IF initializeEvents THEN 
	initializeEvents := FALSE; 
	Emergency_zone_1.CreateEx(TC_Events.Kremer_Events.Emergency_zone_1, TRUE, 0); 
	Emergency_zone_2.CreateEx(TC_Events.Kremer_Events.Emergency_zone_2, TRUE, 0); 
	Emergency_zone_3.CreateEx(TC_Events.Kremer_Events.Emergency_zone_3, TRUE, 0); 
	Emergency_zone_4.CreateEx(TC_Events.Kremer_Events.Emergency_zone_4, TRUE, 0); 
	Emergency_zone_5.CreateEx(TC_Events.Kremer_Events.Emergency_zone_5, TRUE, 0); 
	Emergency_zone_6.CreateEx(TC_Events.Kremer_Events.Emergency_zone_6, TRUE, 0); 
	Emergency_zone_7.CreateEx(TC_Events.Kremer_Events.Emergency_zone_7, TRUE, 0); 
	In_mold_drying_emergency_stop_pressed_front_side.CreateEx(TC_Events.Kremer_Events.In_mold_drying_emergency_stop_pressed_front_side, TRUE, 0); 
	In_mold_drying_emergency_stop_pressed_back_side.CreateEx(TC_Events.Kremer_Events.In_mold_drying_emergency_stop_pressed_back_side, TRUE, 0); 
	In_mold_drying_door_opend_frontside_left.CreateEx(TC_Events.Kremer_Events.In_mold_drying_door_opend_frontside_left, TRUE, 0); 
	In_mold_drying_door_opened_frontside_middle.CreateEx(TC_Events.Kremer_Events.In_mold_drying_door_opened_frontside_middle, TRUE, 0); 
	In_mold_drying_door_opened_frontside_right.CreateEx(TC_Events.Kremer_Events.In_mold_drying_door_opened_frontside_right, TRUE, 0); 
	In_mold_drying_double_door_opened_backside_left_1.CreateEx(TC_Events.Kremer_Events.In_mold_drying_double_door_opened_backside_left_1, TRUE, 0); 
	In_mold_drying_double_door_opened_backside_left_2.CreateEx(TC_Events.Kremer_Events.In_mold_drying_double_door_opened_backside_left_2, TRUE, 0); 
	In_mold_drying_double_door_opened_backside_Middle_1.CreateEx(TC_Events.Kremer_Events.In_mold_drying_double_door_opened_backside_Middle_1, TRUE, 0); 
	In_mold_drying_double_door_opened_backside_Middle_2.CreateEx(TC_Events.Kremer_Events.In_mold_drying_double_door_opened_backside_Middle_2, TRUE, 0); 
	In_mold_drying_double_door_opened_backside_Right_1.CreateEx(TC_Events.Kremer_Events.In_mold_drying_double_door_opened_backside_Right_1, TRUE, 0); 
	In_mold_drying_double_door_opened_backside_Right_2.CreateEx(TC_Events.Kremer_Events.In_mold_drying_double_door_opened_backside_Right_2, TRUE, 0); 
	Gantry_A_front_door_openend_right.CreateEx(TC_Events.Kremer_Events.Gantry_A_front_door_openend_right, TRUE, 0); 
	Gantry_A_front_door_openend_left.CreateEx(TC_Events.Kremer_Events.Gantry_A_front_door_openend_left, TRUE, 0); 
	Gantry_A_Back_door_openend.CreateEx(TC_Events.Kremer_Events.Gantry_A_Back_door_openend, TRUE, 0); 
	Gantry_B_front_door_openend_left.CreateEx(TC_Events.Kremer_Events.Gantry_B_front_door_openend_left, TRUE, 0); 
	Gantry_B_front_door_openend_right.CreateEx(TC_Events.Kremer_Events.Gantry_B_front_door_openend_right, TRUE, 0); 
	Gantry_B_Back_door_openend.CreateEx(TC_Events.Kremer_Events.Gantry_B_Back_door_openend, TRUE, 0); 
	Emergency_stop_pressed_Gantry_A_backside.CreateEx(TC_Events.Kremer_Events.Emergency_stop_pressed_Gantry_A_backside, TRUE, 0); 
	Emergency_stop_pressed_Gantry_A_Frontside.CreateEx(TC_Events.Kremer_Events.Emergency_stop_pressed_Gantry_A_Frontside, TRUE, 0); 
	Emergency_stop_pressed_Gantry_B_Backside.CreateEx(TC_Events.Kremer_Events.Emergency_stop_pressed_Gantry_B_Backside, TRUE, 0); 
	Emergency_stop_pressed_Gantry_B_Frontside.CreateEx(TC_Events.Kremer_Events.Emergency_stop_pressed_Gantry_B_Frontside, TRUE, 0); 
	_24_volt_circuit_in_error_1.CreateEx(TC_Events.Kremer_Events._24_volt_circuit_in_error_1, TRUE, 0); 
	_24_volt_circuit_in_error_2.CreateEx(TC_Events.Kremer_Events._24_volt_circuit_in_error_2, TRUE, 0); 
	No_product_loaded_please_load_a_valid_product_first.CreateEx(TC_Events.Kremer_Events.No_product_loaded_please_load_a_valid_product_first, TRUE, 0); 
	Main_air_supply_has_an_error.CreateEx(TC_Events.Kremer_Events.Main_air_supply_has_an_error, TRUE, 0); 
	In_mold_drying_hydraulic_pump_softstarter_failure.CreateEx(TC_Events.Kremer_Events.In_mold_drying_hydraulic_pump_softstarter_failure, TRUE, 0); 
	In_mold_drying_hydraulic_pump_maintenance_switch.CreateEx(TC_Events.Kremer_Events.In_mold_drying_hydraulic_pump_maintenance_switch, TRUE, 0); 
	In_mold_drying_cooling_fan_thermal_failure.CreateEx(TC_Events.Kremer_Events.In_mold_drying_cooling_fan_thermal_failure, TRUE, 0); 
	In_mold_drying_cooling_fan_maintenance_switch.CreateEx(TC_Events.Kremer_Events.In_mold_drying_cooling_fan_maintenance_switch, TRUE, 0); 
	In_mold_drying_filter_motor_thermal.CreateEx(TC_Events.Kremer_Events.In_mold_drying_filter_motor_thermal, TRUE, 0); 
	In_mold_drying_filter_motor_maintenance.CreateEx(TC_Events.Kremer_Events.In_mold_drying_filter_motor_maintenance, TRUE, 0); 
	Css_has_an_active_error.CreateEx(TC_Events.Kremer_Events.Css_has_an_active_error, TRUE, 0); 
	Both_Pulp_Tanks_below_Low_Level_stopping_IMD.CreateEx(TC_Events.Kremer_Events.Both_Pulp_Tanks_below_Low_Level_stopping_IMD, TRUE, 0); 
	RHSR_Bottom_mold_A_moving_while_top_mold_A_not_in_position.CreateEx(TC_Events.Kremer_Events.RHSR_Bottom_mold_A_moving_while_top_mold_A_not_in_position, TRUE, 0); 
	RHSR_Bottom_mold_A_moving_while_transfer_mold_A_not_in_position.CreateEx(TC_Events.Kremer_Events.RHSR_Bottom_mold_A_moving_while_transfer_mold_A_not_in_position, TRUE, 0); 
	RHSR_Bottom_mold_B_moving_while_top_mold_B_not_in_position.CreateEx(TC_Events.Kremer_Events.RHSR_Bottom_mold_B_moving_while_top_mold_B_not_in_position, TRUE, 0); 
	RHSR_Bottom_mold_B_moving_while_transfer_mold_B_not_in_position.CreateEx(TC_Events.Kremer_Events.RHSR_Bottom_mold_B_moving_while_transfer_mold_B_not_in_position, TRUE, 0); 
	RHSR_Takeout_A_moving_while_vertical_cylinder_is_not_down.CreateEx(TC_Events.Kremer_Events.RHSR_Takeout_A_moving_while_vertical_cylinder_is_not_down, TRUE, 0); 
	RHSR_Takeout_B_moving_while_vertical_cylinder_is_not_down.CreateEx(TC_Events.Kremer_Events.RHSR_Takeout_B_moving_while_vertical_cylinder_is_not_down, TRUE, 0); 
	RHSR_TopMold_A_moving_while_bottom_mold_A_is_not_in_position.CreateEx(TC_Events.Kremer_Events.RHSR_TopMold_A_moving_while_bottom_mold_A_is_not_in_position, TRUE, 0); 
	RHSR_TopMold_B_moving_while_bottom_mold_B_is_not_in_position.CreateEx(TC_Events.Kremer_Events.RHSR_TopMold_B_moving_while_bottom_mold_B_is_not_in_position, TRUE, 0); 
	RHSR_Transfermold_moving_while_bottom_mold_A_is_not_in_posititon.CreateEx(TC_Events.Kremer_Events.RHSR_Transfermold_moving_while_bottom_mold_A_is_not_in_posititon, TRUE, 0); 
	RHSR_Transfermold_moving_while_bottom_mold_B_is_not_in_position.CreateEx(TC_Events.Kremer_Events.RHSR_Transfermold_moving_while_bottom_mold_B_is_not_in_position, TRUE, 0); 
	RHSR_Transfermold_moving_while_spraybar_is_not_at_one_of_rest_positions.CreateEx(TC_Events.Kremer_Events.RHSR_Transfermold_moving_while_spraybar_is_not_at_one_of_rest_positions, TRUE, 0); 
	Temperature_difference_between_top_and_bottom_mold_side_A_to_high.CreateEx(TC_Events.Kremer_Events.Temperature_difference_between_top_and_bottom_mold_side_A_to_high, TRUE, 0); 
	Temperature_difference_between_top_and_bottom_mold_side_B_to_high.CreateEx(TC_Events.Kremer_Events.Temperature_difference_between_top_and_bottom_mold_side_B_to_high, TRUE, 0); 
	Spare56.CreateEx(TC_Events.Kremer_Events.Spare56, TRUE, 0); 
	Auxiliary_filter_100_dirty.CreateEx(TC_Events.Kremer_Events.Auxiliary_filter_100_dirty, TRUE, 0); 
	Auxiliary_filter_75_dirty.CreateEx(TC_Events.Kremer_Events.Auxiliary_filter_75_dirty, TRUE, 0); 
	Oil_filter_100_dirty.CreateEx(TC_Events.Kremer_Events.Oil_filter_100_dirty, TRUE, 0); 
	Oil_filter_75_dirty.CreateEx(TC_Events.Kremer_Events.Oil_filter_75_dirty, TRUE, 0); 
	Fan_on_MCC2_error.CreateEx(TC_Events.Kremer_Events.Fan_on_MCC2_error, TRUE, 0); 
	_24V_error_on_MCC2.CreateEx(TC_Events.Kremer_Events._24V_error_on_MCC2, TRUE, 0); 
	Oil_temperature_too_low.CreateEx(TC_Events.Kremer_Events.Oil_temperature_too_low, TRUE, 0); 
	Oil_temperature_too_high.CreateEx(TC_Events.Kremer_Events.Oil_temperature_too_high, TRUE, 0); 
	Top_mold_A_error_on_balluf.CreateEx(TC_Events.Kremer_Events.Top_mold_A_error_on_balluf, TRUE, 0); 
	Top_mold_A_position_error.CreateEx(TC_Events.Kremer_Events.Top_mold_A_position_error, TRUE, 0); 
	Top_mold_A_timed_out_Did_not_reach_bottommold_position_in_time.CreateEx(TC_Events.Kremer_Events.Top_mold_A_timed_out_Did_not_reach_bottommold_position_in_time, TRUE, 0); 
	Top_mold_A_Rod_side_pressure_too_high.CreateEx(TC_Events.Kremer_Events.Top_mold_A_Rod_side_pressure_too_high, TRUE, 0); 
	Top_mold_A_Bot_side_pressure_too_high.CreateEx(TC_Events.Kremer_Events.Top_mold_A_Bot_side_pressure_too_high, TRUE, 0); 
	Topmold_A_heating_zone_1_connector_not_connected.CreateEx(TC_Events.Kremer_Events.Topmold_A_heating_zone_1_connector_not_connected, TRUE, 0); 
	Topmold_A_heating_zone_1_PT100_wrong_position.CreateEx(TC_Events.Kremer_Events.Topmold_A_heating_zone_1_PT100_wrong_position, TRUE, 0); 
	Topmold_A_heating_zone_1_PT100_loose.CreateEx(TC_Events.Kremer_Events.Topmold_A_heating_zone_1_PT100_loose, TRUE, 0); 
	Topmold_A_heating_zone_1_PT100_not_inserted.CreateEx(TC_Events.Kremer_Events.Topmold_A_heating_zone_1_PT100_not_inserted, TRUE, 0); 
	Topmold_A_heating_zone_1_Temperature_above_setpoint.CreateEx(TC_Events.Kremer_Events.Topmold_A_heating_zone_1_Temperature_above_setpoint, TRUE, 0); 
	Topmold_A_heating_zone_1_Temperature_below_setpoint.CreateEx(TC_Events.Kremer_Events.Topmold_A_heating_zone_1_Temperature_below_setpoint, TRUE, 0); 
	Topmold_A_heating_zone_1_PT100_wirebreak.CreateEx(TC_Events.Kremer_Events.Topmold_A_heating_zone_1_PT100_wirebreak, TRUE, 0); 
	Topmold_A_heating_zone_1_Thermal.CreateEx(TC_Events.Kremer_Events.Topmold_A_heating_zone_1_Thermal, TRUE, 0); 
	Topmold_A_heating_zone_1_temperature_above_250_degree_heating_element_switched_off.CreateEx(TC_Events.Kremer_Events.Topmold_A_heating_zone_1_temperature_above_250_degree_heating_element_switched_off, TRUE, 0); 
	Topmold_A_heating_zone_1_temperature_above_230_degree.CreateEx(TC_Events.Kremer_Events.Topmold_A_heating_zone_1_temperature_above_230_degree, TRUE, 0); 
	Topmold_A_heating_zone_2_connector_not_connected.CreateEx(TC_Events.Kremer_Events.Topmold_A_heating_zone_2_connector_not_connected, TRUE, 0); 
	Topmold_A_heating_zone_2_PT100_wrong_position.CreateEx(TC_Events.Kremer_Events.Topmold_A_heating_zone_2_PT100_wrong_position, TRUE, 0); 
	Topmold_A_heating_zone_2_PT100_loose.CreateEx(TC_Events.Kremer_Events.Topmold_A_heating_zone_2_PT100_loose, TRUE, 0); 
	Topmold_A_heating_zone_2_PT100_not_inserted.CreateEx(TC_Events.Kremer_Events.Topmold_A_heating_zone_2_PT100_not_inserted, TRUE, 0); 
	Topmold_A_heating_zone_2_Temperature_above_setpoint.CreateEx(TC_Events.Kremer_Events.Topmold_A_heating_zone_2_Temperature_above_setpoint, TRUE, 0); 
	Topmold_A_heating_zone_2_Temperature_below_setpoint.CreateEx(TC_Events.Kremer_Events.Topmold_A_heating_zone_2_Temperature_below_setpoint, TRUE, 0); 
	Topmold_A_heating_zone_2_PT100_wirebreak.CreateEx(TC_Events.Kremer_Events.Topmold_A_heating_zone_2_PT100_wirebreak, TRUE, 0); 
	Topmold_A_heating_zone_2_Thermal.CreateEx(TC_Events.Kremer_Events.Topmold_A_heating_zone_2_Thermal, TRUE, 0); 
	Topmold_A_heating_zone_2_temperature_above_250_degree_heating_element_switched_off.CreateEx(TC_Events.Kremer_Events.Topmold_A_heating_zone_2_temperature_above_250_degree_heating_element_switched_off, TRUE, 0); 
	Topmold_A_heating_zone_2_temperature_above_230_degree.CreateEx(TC_Events.Kremer_Events.Topmold_A_heating_zone_2_temperature_above_230_degree, TRUE, 0); 
	Tranfermold_timed_out_did_not_reach_bottommold_position_in_time.CreateEx(TC_Events.Kremer_Events.Tranfermold_timed_out_did_not_reach_bottommold_position_in_time, TRUE, 0); 
	Tranfermold_timed_out_did_not_reach_forming_position_in_time.CreateEx(TC_Events.Kremer_Events.Tranfermold_timed_out_did_not_reach_forming_position_in_time, TRUE, 0); 
	Topmold_A_heating_zone_3_connector_not_connected.CreateEx(TC_Events.Kremer_Events.Topmold_A_heating_zone_3_connector_not_connected, TRUE, 0); 
	Topmold_A_heating_zone_3_PT100_wrong_position.CreateEx(TC_Events.Kremer_Events.Topmold_A_heating_zone_3_PT100_wrong_position, TRUE, 0); 
	Topmold_A_heating_zone_3_PT100_loose.CreateEx(TC_Events.Kremer_Events.Topmold_A_heating_zone_3_PT100_loose, TRUE, 0); 
	Topmold_A_heating_zone_3_PT100_not_inserted.CreateEx(TC_Events.Kremer_Events.Topmold_A_heating_zone_3_PT100_not_inserted, TRUE, 0); 
	Topmold_A_heating_zone_3_Temperature_above_setpoint.CreateEx(TC_Events.Kremer_Events.Topmold_A_heating_zone_3_Temperature_above_setpoint, TRUE, 0); 
	Topmold_A_heating_zone_3_Temperature_below_setpoint.CreateEx(TC_Events.Kremer_Events.Topmold_A_heating_zone_3_Temperature_below_setpoint, TRUE, 0); 
	Topmold_A_heating_zone_3_PT100_wirebreak.CreateEx(TC_Events.Kremer_Events.Topmold_A_heating_zone_3_PT100_wirebreak, TRUE, 0); 
	Topmold_A_heating_zone_3_Thermal.CreateEx(TC_Events.Kremer_Events.Topmold_A_heating_zone_3_Thermal, TRUE, 0); 
	Topmold_A_heating_zone_3_temperature_above_250_degree_heating_element_switched_off.CreateEx(TC_Events.Kremer_Events.Topmold_A_heating_zone_3_temperature_above_250_degree_heating_element_switched_off, TRUE, 0); 
	Topmold_A_heating_zone_3_temperature_above_230_degree.CreateEx(TC_Events.Kremer_Events.Topmold_A_heating_zone_3_temperature_above_230_degree, TRUE, 0); 
	Topmold_A_heating_zone_4_connector_not_connected.CreateEx(TC_Events.Kremer_Events.Topmold_A_heating_zone_4_connector_not_connected, TRUE, 0); 
	Topmold_A_heating_zone_4_PT100_wrong_position.CreateEx(TC_Events.Kremer_Events.Topmold_A_heating_zone_4_PT100_wrong_position, TRUE, 0); 
	Topmold_A_heating_zone_4_PT100_loose.CreateEx(TC_Events.Kremer_Events.Topmold_A_heating_zone_4_PT100_loose, TRUE, 0); 
	Topmold_A_heating_zone_4_PT100_not_inserted.CreateEx(TC_Events.Kremer_Events.Topmold_A_heating_zone_4_PT100_not_inserted, TRUE, 0); 
	Topmold_A_heating_zone_4_Temperature_above_setpoint.CreateEx(TC_Events.Kremer_Events.Topmold_A_heating_zone_4_Temperature_above_setpoint, TRUE, 0); 
	Topmold_A_heating_zone_4_Temperature_below_setpoint.CreateEx(TC_Events.Kremer_Events.Topmold_A_heating_zone_4_Temperature_below_setpoint, TRUE, 0); 
	Topmold_A_heating_zone_4_PT100_wirebreak.CreateEx(TC_Events.Kremer_Events.Topmold_A_heating_zone_4_PT100_wirebreak, TRUE, 0); 
	Topmold_A_heating_zone_4_Thermal.CreateEx(TC_Events.Kremer_Events.Topmold_A_heating_zone_4_Thermal, TRUE, 0); 
	Topmold_A_heating_zone_4_temperature_above_250_degree_heating_element_switched_off.CreateEx(TC_Events.Kremer_Events.Topmold_A_heating_zone_4_temperature_above_250_degree_heating_element_switched_off, TRUE, 0); 
	Topmold_A_heating_zone_4_temperature_above_230_degree.CreateEx(TC_Events.Kremer_Events.Topmold_A_heating_zone_4_temperature_above_230_degree, TRUE, 0); 
	Topmold_A_heating_zone_5_connector_not_connected.CreateEx(TC_Events.Kremer_Events.Topmold_A_heating_zone_5_connector_not_connected, TRUE, 0); 
	Topmold_A_heating_zone_5_PT100_wrong_position.CreateEx(TC_Events.Kremer_Events.Topmold_A_heating_zone_5_PT100_wrong_position, TRUE, 0); 
	Topmold_A_heating_zone_5_PT100_loose.CreateEx(TC_Events.Kremer_Events.Topmold_A_heating_zone_5_PT100_loose, TRUE, 0); 
	Topmold_A_heating_zone_5_PT100_not_inserted.CreateEx(TC_Events.Kremer_Events.Topmold_A_heating_zone_5_PT100_not_inserted, TRUE, 0); 
	Topmold_A_heating_zone_5_Temperature_above_setpoint.CreateEx(TC_Events.Kremer_Events.Topmold_A_heating_zone_5_Temperature_above_setpoint, TRUE, 0); 
	Topmold_A_heating_zone_5_Temperature_below_setpoint.CreateEx(TC_Events.Kremer_Events.Topmold_A_heating_zone_5_Temperature_below_setpoint, TRUE, 0); 
	Topmold_A_heating_zone_5_PT100_wirebreak.CreateEx(TC_Events.Kremer_Events.Topmold_A_heating_zone_5_PT100_wirebreak, TRUE, 0); 
	Topmold_A_heating_zone_5_Thermal.CreateEx(TC_Events.Kremer_Events.Topmold_A_heating_zone_5_Thermal, TRUE, 0); 
	Topmold_A_heating_zone_5_temperature_above_250_degree_heating_element_switched_off.CreateEx(TC_Events.Kremer_Events.Topmold_A_heating_zone_5_temperature_above_250_degree_heating_element_switched_off, TRUE, 0); 
	Topmold_A_heating_zone_5_temperature_above_230_degree.CreateEx(TC_Events.Kremer_Events.Topmold_A_heating_zone_5_temperature_above_230_degree, TRUE, 0); 
	Topmold_A_heating_zone_6_connector_not_connected.CreateEx(TC_Events.Kremer_Events.Topmold_A_heating_zone_6_connector_not_connected, TRUE, 0); 
	Topmold_A_heating_zone_6_PT100_wrong_position.CreateEx(TC_Events.Kremer_Events.Topmold_A_heating_zone_6_PT100_wrong_position, TRUE, 0); 
	Topmold_A_heating_zone_6_PT100_loose.CreateEx(TC_Events.Kremer_Events.Topmold_A_heating_zone_6_PT100_loose, TRUE, 0); 
	Topmold_A_heating_zone_6_PT100_not_inserted.CreateEx(TC_Events.Kremer_Events.Topmold_A_heating_zone_6_PT100_not_inserted, TRUE, 0); 
	Topmold_A_heating_zone_6_Temperature_above_setpoint.CreateEx(TC_Events.Kremer_Events.Topmold_A_heating_zone_6_Temperature_above_setpoint, TRUE, 0); 
	Topmold_A_heating_zone_6_Temperature_below_setpoint.CreateEx(TC_Events.Kremer_Events.Topmold_A_heating_zone_6_Temperature_below_setpoint, TRUE, 0); 
	Topmold_A_heating_zone_6_PT100_wirebreak.CreateEx(TC_Events.Kremer_Events.Topmold_A_heating_zone_6_PT100_wirebreak, TRUE, 0); 
	Topmold_A_heating_zone_6_Thermal.CreateEx(TC_Events.Kremer_Events.Topmold_A_heating_zone_6_Thermal, TRUE, 0); 
	Topmold_A_heating_zone_6_temperature_above_250_degree_heating_element_switched_off.CreateEx(TC_Events.Kremer_Events.Topmold_A_heating_zone_6_temperature_above_250_degree_heating_element_switched_off, TRUE, 0); 
	Topmold_A_heating_zone_6_temperature_above_230_degree.CreateEx(TC_Events.Kremer_Events.Topmold_A_heating_zone_6_temperature_above_230_degree, TRUE, 0); 
	Bottommold_A_heating_Zone_1_connector_not_connected.CreateEx(TC_Events.Kremer_Events.Bottommold_A_heating_Zone_1_connector_not_connected, TRUE, 0); 
	Bottommold_A_heating_Zone_1_PT100_wrong_position.CreateEx(TC_Events.Kremer_Events.Bottommold_A_heating_Zone_1_PT100_wrong_position, TRUE, 0); 
	Bottommold_A_heating_Zone_1_PT100_loose.CreateEx(TC_Events.Kremer_Events.Bottommold_A_heating_Zone_1_PT100_loose, TRUE, 0); 
	Bottommold_A_heating_Zone_1_PT100_not_inserted.CreateEx(TC_Events.Kremer_Events.Bottommold_A_heating_Zone_1_PT100_not_inserted, TRUE, 0); 
	Bottommold_A_heating_Zone_1_Temperature_above_setpoint.CreateEx(TC_Events.Kremer_Events.Bottommold_A_heating_Zone_1_Temperature_above_setpoint, TRUE, 0); 
	Bottommold_A_heating_Zone_1_Temperature_below_setpoint.CreateEx(TC_Events.Kremer_Events.Bottommold_A_heating_Zone_1_Temperature_below_setpoint, TRUE, 0); 
	Bottommold_A_heating_Zone_1_PT100_wirebreak.CreateEx(TC_Events.Kremer_Events.Bottommold_A_heating_Zone_1_PT100_wirebreak, TRUE, 0); 
	Bottommold_A_heating_Zone_1_Thermal.CreateEx(TC_Events.Kremer_Events.Bottommold_A_heating_Zone_1_Thermal, TRUE, 0); 
	Bottommold_A_heating_zone_1_temperature_above_250_degree_heating_element_switched_off.CreateEx(TC_Events.Kremer_Events.Bottommold_A_heating_zone_1_temperature_above_250_degree_heating_element_switched_off, TRUE, 0); 
	Bottommold_A_heating_zone_1_temperature_above_230_degree.CreateEx(TC_Events.Kremer_Events.Bottommold_A_heating_zone_1_temperature_above_230_degree, TRUE, 0); 
	Bottommold_A_heating_Zone_2_connector_not_connected.CreateEx(TC_Events.Kremer_Events.Bottommold_A_heating_Zone_2_connector_not_connected, TRUE, 0); 
	Bottommold_A_heating_Zone_2_PT100_wrong_position.CreateEx(TC_Events.Kremer_Events.Bottommold_A_heating_Zone_2_PT100_wrong_position, TRUE, 0); 
	Bottommold_A_heating_Zone_2_PT100_loose.CreateEx(TC_Events.Kremer_Events.Bottommold_A_heating_Zone_2_PT100_loose, TRUE, 0); 
	Bottommold_A_heating_Zone_2_PT100_not_inserted.CreateEx(TC_Events.Kremer_Events.Bottommold_A_heating_Zone_2_PT100_not_inserted, TRUE, 0); 
	Bottommold_A_heating_Zone_2_Temperature_above_setpoint.CreateEx(TC_Events.Kremer_Events.Bottommold_A_heating_Zone_2_Temperature_above_setpoint, TRUE, 0); 
	Bottommold_A_heating_Zone_2_Temperature_below_setpoint.CreateEx(TC_Events.Kremer_Events.Bottommold_A_heating_Zone_2_Temperature_below_setpoint, TRUE, 0); 
	Bottommold_A_heating_Zone_2_PT100_wirebreak.CreateEx(TC_Events.Kremer_Events.Bottommold_A_heating_Zone_2_PT100_wirebreak, TRUE, 0); 
	Bottommold_A_heating_Zone_2_Thermal.CreateEx(TC_Events.Kremer_Events.Bottommold_A_heating_Zone_2_Thermal, TRUE, 0); 
	Bottommold_A_heating_zone_2_temperature_above_250_degree_heating_element_switched_off.CreateEx(TC_Events.Kremer_Events.Bottommold_A_heating_zone_2_temperature_above_250_degree_heating_element_switched_off, TRUE, 0); 
	Bottommold_A_heating_zone_2_temperature_above_230_degree.CreateEx(TC_Events.Kremer_Events.Bottommold_A_heating_zone_2_temperature_above_230_degree, TRUE, 0); 
	Bottommold_A_heating_Zone_3_connector_not_connected.CreateEx(TC_Events.Kremer_Events.Bottommold_A_heating_Zone_3_connector_not_connected, TRUE, 0); 
	Bottommold_A_heating_Zone_3_PT100_wrong_position.CreateEx(TC_Events.Kremer_Events.Bottommold_A_heating_Zone_3_PT100_wrong_position, TRUE, 0); 
	Bottommold_A_heating_Zone_3_PT100_loose.CreateEx(TC_Events.Kremer_Events.Bottommold_A_heating_Zone_3_PT100_loose, TRUE, 0); 
	Bottommold_A_heating_Zone_3_PT100_not_inserted.CreateEx(TC_Events.Kremer_Events.Bottommold_A_heating_Zone_3_PT100_not_inserted, TRUE, 0); 
	Bottommold_A_heating_Zone_3_Temperature_above_setpoint.CreateEx(TC_Events.Kremer_Events.Bottommold_A_heating_Zone_3_Temperature_above_setpoint, TRUE, 0); 
	Bottommold_A_heating_Zone_3_Temperature_below_setpoint.CreateEx(TC_Events.Kremer_Events.Bottommold_A_heating_Zone_3_Temperature_below_setpoint, TRUE, 0); 
	Bottommold_A_heating_Zone_3_PT100_wirebreak.CreateEx(TC_Events.Kremer_Events.Bottommold_A_heating_Zone_3_PT100_wirebreak, TRUE, 0); 
	Bottommold_A_heating_Zone_3_Thermal.CreateEx(TC_Events.Kremer_Events.Bottommold_A_heating_Zone_3_Thermal, TRUE, 0); 
	Bottommold_A_heating_zone_3_temperature_above_250_degree_heating_element_switched_off.CreateEx(TC_Events.Kremer_Events.Bottommold_A_heating_zone_3_temperature_above_250_degree_heating_element_switched_off, TRUE, 0); 
	Bottommold_A_heating_zone_3_temperature_above_230_degree.CreateEx(TC_Events.Kremer_Events.Bottommold_A_heating_zone_3_temperature_above_230_degree, TRUE, 0); 
	Bottommold_A_heating_Zone_4_connector_not_connected.CreateEx(TC_Events.Kremer_Events.Bottommold_A_heating_Zone_4_connector_not_connected, TRUE, 0); 
	Bottommold_A_heating_Zone_4_PT100_wrong_position.CreateEx(TC_Events.Kremer_Events.Bottommold_A_heating_Zone_4_PT100_wrong_position, TRUE, 0); 
	Bottommold_A_heating_Zone_4_PT100_loose.CreateEx(TC_Events.Kremer_Events.Bottommold_A_heating_Zone_4_PT100_loose, TRUE, 0); 
	Bottommold_A_heating_Zone_4_PT100_not_inserted.CreateEx(TC_Events.Kremer_Events.Bottommold_A_heating_Zone_4_PT100_not_inserted, TRUE, 0); 
	Bottommold_A_heating_Zone_4_Temperature_above_setpoint.CreateEx(TC_Events.Kremer_Events.Bottommold_A_heating_Zone_4_Temperature_above_setpoint, TRUE, 0); 
	Bottommold_A_heating_Zone_4_Temperature_below_setpoint.CreateEx(TC_Events.Kremer_Events.Bottommold_A_heating_Zone_4_Temperature_below_setpoint, TRUE, 0); 
	Bottommold_A_heating_Zone_4_PT100_wirebreak.CreateEx(TC_Events.Kremer_Events.Bottommold_A_heating_Zone_4_PT100_wirebreak, TRUE, 0); 
	Bottommold_A_heating_Zone_4_Thermal.CreateEx(TC_Events.Kremer_Events.Bottommold_A_heating_Zone_4_Thermal, TRUE, 0); 
	Bottommold_A_heating_zone_4_temperature_above_250_degree_heating_element_switched_off.CreateEx(TC_Events.Kremer_Events.Bottommold_A_heating_zone_4_temperature_above_250_degree_heating_element_switched_off, TRUE, 0); 
	Bottommold_A_heating_zone_4_temperature_above_230_degree.CreateEx(TC_Events.Kremer_Events.Bottommold_A_heating_zone_4_temperature_above_230_degree, TRUE, 0); 
	Bottommold_A_heating_Zone_5_connector_not_connected.CreateEx(TC_Events.Kremer_Events.Bottommold_A_heating_Zone_5_connector_not_connected, TRUE, 0); 
	Bottommold_A_heating_Zone_5_PT100_wrong_position.CreateEx(TC_Events.Kremer_Events.Bottommold_A_heating_Zone_5_PT100_wrong_position, TRUE, 0); 
	Bottommold_A_heating_Zone_5_PT100_loose.CreateEx(TC_Events.Kremer_Events.Bottommold_A_heating_Zone_5_PT100_loose, TRUE, 0); 
	Bottommold_A_heating_Zone_5_PT100_not_inserted.CreateEx(TC_Events.Kremer_Events.Bottommold_A_heating_Zone_5_PT100_not_inserted, TRUE, 0); 
	Bottommold_A_heating_Zone_5_Temperature_above_setpoint.CreateEx(TC_Events.Kremer_Events.Bottommold_A_heating_Zone_5_Temperature_above_setpoint, TRUE, 0); 
	Bottommold_A_heating_Zone_5_Temperature_below_setpoint.CreateEx(TC_Events.Kremer_Events.Bottommold_A_heating_Zone_5_Temperature_below_setpoint, TRUE, 0); 
	Bottommold_A_heating_Zone_5_PT100_wirebreak.CreateEx(TC_Events.Kremer_Events.Bottommold_A_heating_Zone_5_PT100_wirebreak, TRUE, 0); 
	Bottommold_A_heating_Zone_5_Thermal.CreateEx(TC_Events.Kremer_Events.Bottommold_A_heating_Zone_5_Thermal, TRUE, 0); 
	Bottommold_A_heating_zone_5_temperature_above_250_degree_heating_element_switched_off.CreateEx(TC_Events.Kremer_Events.Bottommold_A_heating_zone_5_temperature_above_250_degree_heating_element_switched_off, TRUE, 0); 
	Bottommold_A_heating_zone_5_temperature_above_230_degree.CreateEx(TC_Events.Kremer_Events.Bottommold_A_heating_zone_5_temperature_above_230_degree, TRUE, 0); 
	Bottommold_A_heating_Zone_6_connector_not_connected.CreateEx(TC_Events.Kremer_Events.Bottommold_A_heating_Zone_6_connector_not_connected, TRUE, 0); 
	Bottommold_A_heating_Zone_6_PT100_wrong_position.CreateEx(TC_Events.Kremer_Events.Bottommold_A_heating_Zone_6_PT100_wrong_position, TRUE, 0); 
	Bottommold_A_heating_Zone_6_PT100_loose.CreateEx(TC_Events.Kremer_Events.Bottommold_A_heating_Zone_6_PT100_loose, TRUE, 0); 
	Bottommold_A_heating_Zone_6_PT100_not_inserted.CreateEx(TC_Events.Kremer_Events.Bottommold_A_heating_Zone_6_PT100_not_inserted, TRUE, 0); 
	Bottommold_A_heating_Zone_6_Temperature_above_setpoint.CreateEx(TC_Events.Kremer_Events.Bottommold_A_heating_Zone_6_Temperature_above_setpoint, TRUE, 0); 
	Bottommold_A_heating_Zone_6_Temperature_below_setpoint.CreateEx(TC_Events.Kremer_Events.Bottommold_A_heating_Zone_6_Temperature_below_setpoint, TRUE, 0); 
	Bottommold_A_heating_Zone_6_PT100_wirebreak.CreateEx(TC_Events.Kremer_Events.Bottommold_A_heating_Zone_6_PT100_wirebreak, TRUE, 0); 
	Bottommold_A_heating_Zone_6_Thermal.CreateEx(TC_Events.Kremer_Events.Bottommold_A_heating_Zone_6_Thermal, TRUE, 0); 
	Bottommold_A_heating_zone_6_temperature_above_250_degree_heating_element_switched_off.CreateEx(TC_Events.Kremer_Events.Bottommold_A_heating_zone_6_temperature_above_250_degree_heating_element_switched_off, TRUE, 0); 
	Top_mold_B_timed_out_Did_not_reach_bottommold_position_in_time.CreateEx(TC_Events.Kremer_Events.Top_mold_B_timed_out_Did_not_reach_bottommold_position_in_time, TRUE, 0); 
	Top_mold_B_error_on_balluf.CreateEx(TC_Events.Kremer_Events.Top_mold_B_error_on_balluf, TRUE, 0); 
	Top_mold_B_is_moving_without_activation.CreateEx(TC_Events.Kremer_Events.Top_mold_B_is_moving_without_activation, TRUE, 0); 
	Bottommold_A_heating_zone_6_temperature_above_230_degree.CreateEx(TC_Events.Kremer_Events.Bottommold_A_heating_zone_6_temperature_above_230_degree, TRUE, 0); 
	Topmold_B_heating_Zone_1_connector_not_connected.CreateEx(TC_Events.Kremer_Events.Topmold_B_heating_Zone_1_connector_not_connected, TRUE, 0); 
	Topmold_B_heating_Zone_1_PT100_wrong_position.CreateEx(TC_Events.Kremer_Events.Topmold_B_heating_Zone_1_PT100_wrong_position, TRUE, 0); 
	Topmold_B_heating_Zone_1_PT100_loose.CreateEx(TC_Events.Kremer_Events.Topmold_B_heating_Zone_1_PT100_loose, TRUE, 0); 
	Topmold_B_heating_Zone_1_PT100_not_inserted.CreateEx(TC_Events.Kremer_Events.Topmold_B_heating_Zone_1_PT100_not_inserted, TRUE, 0); 
	Topmold_B_heating_Zone_1_Temperature_above_setpoint.CreateEx(TC_Events.Kremer_Events.Topmold_B_heating_Zone_1_Temperature_above_setpoint, TRUE, 0); 
	Topmold_B_heating_Zone_1_Temperature_below_setpoint.CreateEx(TC_Events.Kremer_Events.Topmold_B_heating_Zone_1_Temperature_below_setpoint, TRUE, 0); 
	Topmold_B_heating_Zone_1_PT100_wirebreak.CreateEx(TC_Events.Kremer_Events.Topmold_B_heating_Zone_1_PT100_wirebreak, TRUE, 0); 
	Topmold_B_heating_Zone_1_Thermal.CreateEx(TC_Events.Kremer_Events.Topmold_B_heating_Zone_1_Thermal, TRUE, 0); 
	Topmold_B_heating_zone_1_temperature_above_250_degree_heating_element_switched_off.CreateEx(TC_Events.Kremer_Events.Topmold_B_heating_zone_1_temperature_above_250_degree_heating_element_switched_off, TRUE, 0); 
	Topmold_B_heating_zone_1_temperature_above_230_degree.CreateEx(TC_Events.Kremer_Events.Topmold_B_heating_zone_1_temperature_above_230_degree, TRUE, 0); 
	Topmold_B_heating_Zone_2_connector_not_connected.CreateEx(TC_Events.Kremer_Events.Topmold_B_heating_Zone_2_connector_not_connected, TRUE, 0); 
	Topmold_B_heating_Zone_2_PT100_wrong_position.CreateEx(TC_Events.Kremer_Events.Topmold_B_heating_Zone_2_PT100_wrong_position, TRUE, 0); 
	Topmold_B_heating_Zone_2_PT100_loose.CreateEx(TC_Events.Kremer_Events.Topmold_B_heating_Zone_2_PT100_loose, TRUE, 0); 
	Topmold_B_heating_Zone_2_PT100_not_inserted.CreateEx(TC_Events.Kremer_Events.Topmold_B_heating_Zone_2_PT100_not_inserted, TRUE, 0); 
	Topmold_B_heating_Zone_2_Temperature_above_setpoint.CreateEx(TC_Events.Kremer_Events.Topmold_B_heating_Zone_2_Temperature_above_setpoint, TRUE, 0); 
	Topmold_B_heating_Zone_2_Temperature_below_setpoint.CreateEx(TC_Events.Kremer_Events.Topmold_B_heating_Zone_2_Temperature_below_setpoint, TRUE, 0); 
	Topmold_B_heating_Zone_2_PT100_wirebreak.CreateEx(TC_Events.Kremer_Events.Topmold_B_heating_Zone_2_PT100_wirebreak, TRUE, 0); 
	Topmold_B_heating_Zone_2_Thermal.CreateEx(TC_Events.Kremer_Events.Topmold_B_heating_Zone_2_Thermal, TRUE, 0); 
	Topmold_B_heating_zone_2_temperature_above_250_degree_heating_element_switched_off.CreateEx(TC_Events.Kremer_Events.Topmold_B_heating_zone_2_temperature_above_250_degree_heating_element_switched_off, TRUE, 0); 
	Topmold_B_heating_zone_2_temperature_above_230_degree.CreateEx(TC_Events.Kremer_Events.Topmold_B_heating_zone_2_temperature_above_230_degree, TRUE, 0); 
	Topmold_B_heating_Zone_3_connector_not_connected.CreateEx(TC_Events.Kremer_Events.Topmold_B_heating_Zone_3_connector_not_connected, TRUE, 0); 
	Topmold_B_heating_Zone_3_PT100_wrong_position.CreateEx(TC_Events.Kremer_Events.Topmold_B_heating_Zone_3_PT100_wrong_position, TRUE, 0); 
	Topmold_B_heating_Zone_3_PT100_loose.CreateEx(TC_Events.Kremer_Events.Topmold_B_heating_Zone_3_PT100_loose, TRUE, 0); 
	Topmold_B_heating_Zone_3_PT100_not_inserted.CreateEx(TC_Events.Kremer_Events.Topmold_B_heating_Zone_3_PT100_not_inserted, TRUE, 0); 
	Topmold_B_heating_Zone_3_Temperature_above_setpoint.CreateEx(TC_Events.Kremer_Events.Topmold_B_heating_Zone_3_Temperature_above_setpoint, TRUE, 0); 
	Topmold_B_heating_Zone_3_Temperature_below_setpoint.CreateEx(TC_Events.Kremer_Events.Topmold_B_heating_Zone_3_Temperature_below_setpoint, TRUE, 0); 
	Topmold_B_heating_Zone_3_PT100_wirebreak.CreateEx(TC_Events.Kremer_Events.Topmold_B_heating_Zone_3_PT100_wirebreak, TRUE, 0); 
	Topmold_B_heating_Zone_3_Thermal.CreateEx(TC_Events.Kremer_Events.Topmold_B_heating_Zone_3_Thermal, TRUE, 0); 
	Topmold_B_heating_zone_3_temperature_above_250_degree_heating_element_switched_off.CreateEx(TC_Events.Kremer_Events.Topmold_B_heating_zone_3_temperature_above_250_degree_heating_element_switched_off, TRUE, 0); 
	Topmold_B_heating_zone_3_temperature_above_230_degree.CreateEx(TC_Events.Kremer_Events.Topmold_B_heating_zone_3_temperature_above_230_degree, TRUE, 0); 
	Topmold_B_heating_Zone_4_connector_not_connected.CreateEx(TC_Events.Kremer_Events.Topmold_B_heating_Zone_4_connector_not_connected, TRUE, 0); 
	Topmold_B_heating_Zone_4_PT100_wrong_position.CreateEx(TC_Events.Kremer_Events.Topmold_B_heating_Zone_4_PT100_wrong_position, TRUE, 0); 
	Topmold_B_heating_Zone_4_PT100_loose.CreateEx(TC_Events.Kremer_Events.Topmold_B_heating_Zone_4_PT100_loose, TRUE, 0); 
	Topmold_B_heating_Zone_4_PT100_not_inserted.CreateEx(TC_Events.Kremer_Events.Topmold_B_heating_Zone_4_PT100_not_inserted, TRUE, 0); 
	Topmold_B_heating_Zone_4_Temperature_above_setpoint.CreateEx(TC_Events.Kremer_Events.Topmold_B_heating_Zone_4_Temperature_above_setpoint, TRUE, 0); 
	Topmold_B_heating_Zone_4_Temperature_below_setpoint.CreateEx(TC_Events.Kremer_Events.Topmold_B_heating_Zone_4_Temperature_below_setpoint, TRUE, 0); 
	Topmold_B_heating_Zone_4_PT100_wirebreak.CreateEx(TC_Events.Kremer_Events.Topmold_B_heating_Zone_4_PT100_wirebreak, TRUE, 0); 
	Topmold_B_heating_Zone_4_Thermal.CreateEx(TC_Events.Kremer_Events.Topmold_B_heating_Zone_4_Thermal, TRUE, 0); 
	Topmold_B_heating_zone_4_temperature_above_250_degree_heating_element_switched_off.CreateEx(TC_Events.Kremer_Events.Topmold_B_heating_zone_4_temperature_above_250_degree_heating_element_switched_off, TRUE, 0); 
	Topmold_B_heating_zone_4_temperature_above_230_degree.CreateEx(TC_Events.Kremer_Events.Topmold_B_heating_zone_4_temperature_above_230_degree, TRUE, 0); 
	Topmold_B_heating_Zone_5_connector_not_connected.CreateEx(TC_Events.Kremer_Events.Topmold_B_heating_Zone_5_connector_not_connected, TRUE, 0); 
	Topmold_B_heating_Zone_5_PT100_wrong_position.CreateEx(TC_Events.Kremer_Events.Topmold_B_heating_Zone_5_PT100_wrong_position, TRUE, 0); 
	Topmold_B_heating_Zone_5_PT100_loose.CreateEx(TC_Events.Kremer_Events.Topmold_B_heating_Zone_5_PT100_loose, TRUE, 0); 
	Topmold_B_heating_Zone_5_PT100_not_inserted.CreateEx(TC_Events.Kremer_Events.Topmold_B_heating_Zone_5_PT100_not_inserted, TRUE, 0); 
	Topmold_B_heating_Zone_5_Temperature_above_setpoint.CreateEx(TC_Events.Kremer_Events.Topmold_B_heating_Zone_5_Temperature_above_setpoint, TRUE, 0); 
	Topmold_B_heating_Zone_5_Temperature_below_setpoint.CreateEx(TC_Events.Kremer_Events.Topmold_B_heating_Zone_5_Temperature_below_setpoint, TRUE, 0); 
	Topmold_B_heating_Zone_5_PT100_wirebreak.CreateEx(TC_Events.Kremer_Events.Topmold_B_heating_Zone_5_PT100_wirebreak, TRUE, 0); 
	Topmold_B_heating_Zone_5_Thermal.CreateEx(TC_Events.Kremer_Events.Topmold_B_heating_Zone_5_Thermal, TRUE, 0); 
	Topmold_B_heating_zone_5_temperature_above_250_degree_heating_element_switched_off.CreateEx(TC_Events.Kremer_Events.Topmold_B_heating_zone_5_temperature_above_250_degree_heating_element_switched_off, TRUE, 0); 
	Topmold_B_heating_zone_5_temperature_above_230_degree.CreateEx(TC_Events.Kremer_Events.Topmold_B_heating_zone_5_temperature_above_230_degree, TRUE, 0); 
	Topmold_B_heating_Zone_6_connector_not_connected.CreateEx(TC_Events.Kremer_Events.Topmold_B_heating_Zone_6_connector_not_connected, TRUE, 0); 
	Topmold_B_heating_Zone_6_PT100_wrong_position.CreateEx(TC_Events.Kremer_Events.Topmold_B_heating_Zone_6_PT100_wrong_position, TRUE, 0); 
	Topmold_B_heating_Zone_6_PT100_loose.CreateEx(TC_Events.Kremer_Events.Topmold_B_heating_Zone_6_PT100_loose, TRUE, 0); 
	Topmold_B_heating_Zone_6_PT100_not_inserted.CreateEx(TC_Events.Kremer_Events.Topmold_B_heating_Zone_6_PT100_not_inserted, TRUE, 0); 
	Topmold_B_heating_Zone_6_Temperature_above_setpoint.CreateEx(TC_Events.Kremer_Events.Topmold_B_heating_Zone_6_Temperature_above_setpoint, TRUE, 0); 
	Topmold_B_heating_Zone_6_Temperature_below_setpoint.CreateEx(TC_Events.Kremer_Events.Topmold_B_heating_Zone_6_Temperature_below_setpoint, TRUE, 0); 
	Topmold_B_heating_Zone_6_PT100_wirebreak.CreateEx(TC_Events.Kremer_Events.Topmold_B_heating_Zone_6_PT100_wirebreak, TRUE, 0); 
	Topmold_B_heating_Zone_6_Thermal.CreateEx(TC_Events.Kremer_Events.Topmold_B_heating_Zone_6_Thermal, TRUE, 0); 
	Topmold_B_heating_zone_6_temperature_above_250_degree_heating_element_switched_off.CreateEx(TC_Events.Kremer_Events.Topmold_B_heating_zone_6_temperature_above_250_degree_heating_element_switched_off, TRUE, 0); 
	Topmold_B_heating_zone_6_temperature_above_230_degree.CreateEx(TC_Events.Kremer_Events.Topmold_B_heating_zone_6_temperature_above_230_degree, TRUE, 0); 
	Bottom_mold_B_error_on_balluf.CreateEx(TC_Events.Kremer_Events.Bottom_mold_B_error_on_balluf, TRUE, 0); 
	Bottom_mold_B_is_moving_without_activation.CreateEx(TC_Events.Kremer_Events.Bottom_mold_B_is_moving_without_activation, TRUE, 0); 
	Top_mold_B_Bot_side_pressure_too_high.CreateEx(TC_Events.Kremer_Events.Top_mold_B_Bot_side_pressure_too_high, TRUE, 0); 
	Top_mold_B_Rot_side_pressure_too_high.CreateEx(TC_Events.Kremer_Events.Top_mold_B_Rot_side_pressure_too_high, TRUE, 0); 
	Bottom_mold_B_heating_Zone_1_connector_not_connected.CreateEx(TC_Events.Kremer_Events.Bottom_mold_B_heating_Zone_1_connector_not_connected, TRUE, 0); 
	Bottom_mold_B_heating_Zone_1_PT100_wrong_position.CreateEx(TC_Events.Kremer_Events.Bottom_mold_B_heating_Zone_1_PT100_wrong_position, TRUE, 0); 
	Bottom_mold_B_heating_Zone_1_PT100_loose.CreateEx(TC_Events.Kremer_Events.Bottom_mold_B_heating_Zone_1_PT100_loose, TRUE, 0); 
	Bottom_mold_B_heating_Zone_1_PT100_not_inserted.CreateEx(TC_Events.Kremer_Events.Bottom_mold_B_heating_Zone_1_PT100_not_inserted, TRUE, 0); 
	Bottom_mold_B_heating_Zone_1_Temperature_above_setpoint.CreateEx(TC_Events.Kremer_Events.Bottom_mold_B_heating_Zone_1_Temperature_above_setpoint, TRUE, 0); 
	Bottom_mold_B_heating_Zone_1_Temperature_below_setpoint.CreateEx(TC_Events.Kremer_Events.Bottom_mold_B_heating_Zone_1_Temperature_below_setpoint, TRUE, 0); 
	Bottom_mold_B_heating_Zone_1_PT100_wirebreak.CreateEx(TC_Events.Kremer_Events.Bottom_mold_B_heating_Zone_1_PT100_wirebreak, TRUE, 0); 
	Bottom_mold_B_heating_Zone_1_Thermal.CreateEx(TC_Events.Kremer_Events.Bottom_mold_B_heating_Zone_1_Thermal, TRUE, 0); 
	Bottom_mold_B_heating_zone_1_temperature_above_250_degree_heating_element_switched_off.CreateEx(TC_Events.Kremer_Events.Bottom_mold_B_heating_zone_1_temperature_above_250_degree_heating_element_switched_off, TRUE, 0); 
	Bottom_mold_B_heating_zone_1_temperature_above_230_degree.CreateEx(TC_Events.Kremer_Events.Bottom_mold_B_heating_zone_1_temperature_above_230_degree, TRUE, 0); 
	Bottom_mold_B_heating_Zone_2_connector_not_connected.CreateEx(TC_Events.Kremer_Events.Bottom_mold_B_heating_Zone_2_connector_not_connected, TRUE, 0); 
	Bottom_mold_B_heating_Zone_2_PT100_wrong_position.CreateEx(TC_Events.Kremer_Events.Bottom_mold_B_heating_Zone_2_PT100_wrong_position, TRUE, 0); 
	Bottom_mold_B_heating_Zone_2_PT100_loose.CreateEx(TC_Events.Kremer_Events.Bottom_mold_B_heating_Zone_2_PT100_loose, TRUE, 0); 
	Bottom_mold_B_heating_Zone_2_PT100_not_inserted.CreateEx(TC_Events.Kremer_Events.Bottom_mold_B_heating_Zone_2_PT100_not_inserted, TRUE, 0); 
	Bottom_mold_B_heating_Zone_2_Temperature_above_setpoint.CreateEx(TC_Events.Kremer_Events.Bottom_mold_B_heating_Zone_2_Temperature_above_setpoint, TRUE, 0); 
	Bottom_mold_B_heating_Zone_2_Temperature_below_setpoint.CreateEx(TC_Events.Kremer_Events.Bottom_mold_B_heating_Zone_2_Temperature_below_setpoint, TRUE, 0); 
	Bottom_mold_B_heating_Zone_2_PT100_wirebreak.CreateEx(TC_Events.Kremer_Events.Bottom_mold_B_heating_Zone_2_PT100_wirebreak, TRUE, 0); 
	Bottom_mold_B_heating_Zone_2_Thermal.CreateEx(TC_Events.Kremer_Events.Bottom_mold_B_heating_Zone_2_Thermal, TRUE, 0); 
	Bottom_mold_B_heating_zone_2_temperature_above_250_degree_heating_element_switched_off.CreateEx(TC_Events.Kremer_Events.Bottom_mold_B_heating_zone_2_temperature_above_250_degree_heating_element_switched_off, TRUE, 0); 
	Bottom_mold_B_heating_zone_2_temperature_above_230_degree.CreateEx(TC_Events.Kremer_Events.Bottom_mold_B_heating_zone_2_temperature_above_230_degree, TRUE, 0); 
	Bottom_mold_B_heating_Zone_3_connector_not_connected.CreateEx(TC_Events.Kremer_Events.Bottom_mold_B_heating_Zone_3_connector_not_connected, TRUE, 0); 
	Bottom_mold_B_heating_Zone_3_PT100_wrong_position.CreateEx(TC_Events.Kremer_Events.Bottom_mold_B_heating_Zone_3_PT100_wrong_position, TRUE, 0); 
	Bottom_mold_B_heating_Zone_3_PT100_loose.CreateEx(TC_Events.Kremer_Events.Bottom_mold_B_heating_Zone_3_PT100_loose, TRUE, 0); 
	Bottom_mold_B_heating_Zone_3_PT100_not_inserted.CreateEx(TC_Events.Kremer_Events.Bottom_mold_B_heating_Zone_3_PT100_not_inserted, TRUE, 0); 
	Bottom_mold_B_heating_Zone_3_Temperature_above_setpoint.CreateEx(TC_Events.Kremer_Events.Bottom_mold_B_heating_Zone_3_Temperature_above_setpoint, TRUE, 0); 
	Bottom_mold_B_heating_Zone_3_Temperature_below_setpoint.CreateEx(TC_Events.Kremer_Events.Bottom_mold_B_heating_Zone_3_Temperature_below_setpoint, TRUE, 0); 
	Bottom_mold_B_heating_Zone_3_PT100_wirebreak.CreateEx(TC_Events.Kremer_Events.Bottom_mold_B_heating_Zone_3_PT100_wirebreak, TRUE, 0); 
	Bottom_mold_B_heating_Zone_3_Thermal.CreateEx(TC_Events.Kremer_Events.Bottom_mold_B_heating_Zone_3_Thermal, TRUE, 0); 
	Bottom_mold_B_heating_zone_3_temperature_above_250_degree_heating_element_switched_off.CreateEx(TC_Events.Kremer_Events.Bottom_mold_B_heating_zone_3_temperature_above_250_degree_heating_element_switched_off, TRUE, 0); 
	Bottom_mold_B_heating_zone_3_temperature_above_230_degree.CreateEx(TC_Events.Kremer_Events.Bottom_mold_B_heating_zone_3_temperature_above_230_degree, TRUE, 0); 
	Bottom_mold_B_heating_Zone_4_connector_not_connected.CreateEx(TC_Events.Kremer_Events.Bottom_mold_B_heating_Zone_4_connector_not_connected, TRUE, 0); 
	Bottom_mold_B_heating_Zone_4_PT100_wrong_position.CreateEx(TC_Events.Kremer_Events.Bottom_mold_B_heating_Zone_4_PT100_wrong_position, TRUE, 0); 
	Bottom_mold_B_heating_Zone_4_PT100_loose.CreateEx(TC_Events.Kremer_Events.Bottom_mold_B_heating_Zone_4_PT100_loose, TRUE, 0); 
	Bottom_mold_B_heating_Zone_4_PT100_not_inserted.CreateEx(TC_Events.Kremer_Events.Bottom_mold_B_heating_Zone_4_PT100_not_inserted, TRUE, 0); 
	Bottom_mold_B_heating_Zone_4_Temperature_above_setpoint.CreateEx(TC_Events.Kremer_Events.Bottom_mold_B_heating_Zone_4_Temperature_above_setpoint, TRUE, 0); 
	Bottom_mold_B_heating_Zone_4_Temperature_below_setpoint.CreateEx(TC_Events.Kremer_Events.Bottom_mold_B_heating_Zone_4_Temperature_below_setpoint, TRUE, 0); 
	Bottom_mold_B_heating_Zone_4_PT100_wirebreak.CreateEx(TC_Events.Kremer_Events.Bottom_mold_B_heating_Zone_4_PT100_wirebreak, TRUE, 0); 
	Bottom_mold_B_heating_Zone_4_Thermal.CreateEx(TC_Events.Kremer_Events.Bottom_mold_B_heating_Zone_4_Thermal, TRUE, 0); 
	Bottom_mold_B_heating_zone_4_temperature_above_250_degree_heating_element_switched_off.CreateEx(TC_Events.Kremer_Events.Bottom_mold_B_heating_zone_4_temperature_above_250_degree_heating_element_switched_off, TRUE, 0); 
	Bottom_mold_B_heating_zone_4_temperature_above_230_degree.CreateEx(TC_Events.Kremer_Events.Bottom_mold_B_heating_zone_4_temperature_above_230_degree, TRUE, 0); 
	Bottom_mold_B_heating_Zone_5_connector_not_connected.CreateEx(TC_Events.Kremer_Events.Bottom_mold_B_heating_Zone_5_connector_not_connected, TRUE, 0); 
	Bottom_mold_B_heating_Zone_5_PT100_wrong_position.CreateEx(TC_Events.Kremer_Events.Bottom_mold_B_heating_Zone_5_PT100_wrong_position, TRUE, 0); 
	Bottom_mold_B_heating_Zone_5_PT100_loose.CreateEx(TC_Events.Kremer_Events.Bottom_mold_B_heating_Zone_5_PT100_loose, TRUE, 0); 
	Bottom_mold_B_heating_Zone_5_PT100_not_inserted.CreateEx(TC_Events.Kremer_Events.Bottom_mold_B_heating_Zone_5_PT100_not_inserted, TRUE, 0); 
	Bottom_mold_B_heating_Zone_5_Temperature_above_setpoint.CreateEx(TC_Events.Kremer_Events.Bottom_mold_B_heating_Zone_5_Temperature_above_setpoint, TRUE, 0); 
	Bottom_mold_B_heating_Zone_5_Temperature_below_setpoint.CreateEx(TC_Events.Kremer_Events.Bottom_mold_B_heating_Zone_5_Temperature_below_setpoint, TRUE, 0); 
	Bottom_mold_B_heating_Zone_5_PT100_wirebreak.CreateEx(TC_Events.Kremer_Events.Bottom_mold_B_heating_Zone_5_PT100_wirebreak, TRUE, 0); 
	Bottom_mold_B_heating_Zone_5_Thermal.CreateEx(TC_Events.Kremer_Events.Bottom_mold_B_heating_Zone_5_Thermal, TRUE, 0); 
	Bottom_mold_B_heating_zone_5_temperature_above_250_degree_heating_element_switched_off.CreateEx(TC_Events.Kremer_Events.Bottom_mold_B_heating_zone_5_temperature_above_250_degree_heating_element_switched_off, TRUE, 0); 
	Bottom_mold_B_heating_zone_5_temperature_above_230_degree.CreateEx(TC_Events.Kremer_Events.Bottom_mold_B_heating_zone_5_temperature_above_230_degree, TRUE, 0); 
	Bottom_mold_B_heating_Zone_6_connector_not_connected.CreateEx(TC_Events.Kremer_Events.Bottom_mold_B_heating_Zone_6_connector_not_connected, TRUE, 0); 
	Bottom_mold_B_heating_Zone_6_PT100_wrong_position.CreateEx(TC_Events.Kremer_Events.Bottom_mold_B_heating_Zone_6_PT100_wrong_position, TRUE, 0); 
	Bottom_mold_B_heating_Zone_6_PT100_loose.CreateEx(TC_Events.Kremer_Events.Bottom_mold_B_heating_Zone_6_PT100_loose, TRUE, 0); 
	Bottom_mold_B_heating_Zone_6_PT100_not_inserted.CreateEx(TC_Events.Kremer_Events.Bottom_mold_B_heating_Zone_6_PT100_not_inserted, TRUE, 0); 
	Bottom_mold_B_heating_Zone_6_Temperature_above_setpoint.CreateEx(TC_Events.Kremer_Events.Bottom_mold_B_heating_Zone_6_Temperature_above_setpoint, TRUE, 0); 
	Bottom_mold_B_heating_Zone_6_Temperature_below_setpoint.CreateEx(TC_Events.Kremer_Events.Bottom_mold_B_heating_Zone_6_Temperature_below_setpoint, TRUE, 0); 
	Bottom_mold_B_heating_Zone_6_PT100_wirebreak.CreateEx(TC_Events.Kremer_Events.Bottom_mold_B_heating_Zone_6_PT100_wirebreak, TRUE, 0); 
	Bottom_mold_B_heating_Zone_6_Thermal.CreateEx(TC_Events.Kremer_Events.Bottom_mold_B_heating_Zone_6_Thermal, TRUE, 0); 
	Bottom_mold_B_heating_zone_6_temperature_above_250_degree_heating_element_switched_off.CreateEx(TC_Events.Kremer_Events.Bottom_mold_B_heating_zone_6_temperature_above_250_degree_heating_element_switched_off, TRUE, 0); 
	Bottom_mold_B_heating_zone_6_temperature_above_230_degree.CreateEx(TC_Events.Kremer_Events.Bottom_mold_B_heating_zone_6_temperature_above_230_degree, TRUE, 0); 
	Takeout_unit_A_horizontal_cylinder_error.CreateEx(TC_Events.Kremer_Events.Takeout_unit_A_horizontal_cylinder_error, TRUE, 0); 
	Takeout_unit_A_horizontal_cylinder_timeout_in.CreateEx(TC_Events.Kremer_Events.Takeout_unit_A_horizontal_cylinder_timeout_in, TRUE, 0); 
	Takeout_unit_A_horizontal_cylinder_timeout_out.CreateEx(TC_Events.Kremer_Events.Takeout_unit_A_horizontal_cylinder_timeout_out, TRUE, 0); 
	Takeout_unit_B_horizontal_cylinder_error.CreateEx(TC_Events.Kremer_Events.Takeout_unit_B_horizontal_cylinder_error, TRUE, 0); 
	Takeout_unit_B_horizontal_cylinder_timeout_in.CreateEx(TC_Events.Kremer_Events.Takeout_unit_B_horizontal_cylinder_timeout_in, TRUE, 0); 
	Takeout_unit_B_horizontal_cylinder_timeout_out.CreateEx(TC_Events.Kremer_Events.Takeout_unit_B_horizontal_cylinder_timeout_out, TRUE, 0); 
	Takeout_unit_A_vertical_cylinder_error.CreateEx(TC_Events.Kremer_Events.Takeout_unit_A_vertical_cylinder_error, TRUE, 0); 
	Takeout_unit_A_vertical_cylinder_timeout_in.CreateEx(TC_Events.Kremer_Events.Takeout_unit_A_vertical_cylinder_timeout_in, TRUE, 0); 
	Takeout_unit_A_vertical_cylinder_timeout_out.CreateEx(TC_Events.Kremer_Events.Takeout_unit_A_vertical_cylinder_timeout_out, TRUE, 0); 
	Takeout_unit_B_vertical_cylinder_error.CreateEx(TC_Events.Kremer_Events.Takeout_unit_B_vertical_cylinder_error, TRUE, 0); 
	Takeout_unit_B_vertical_cylinder_timeout_in.CreateEx(TC_Events.Kremer_Events.Takeout_unit_B_vertical_cylinder_timeout_in, TRUE, 0); 
	Takeout_unit_B_vertical_cylinder_timeout_out.CreateEx(TC_Events.Kremer_Events.Takeout_unit_B_vertical_cylinder_timeout_out, TRUE, 0); 
	Takeout_unit_A_error_on_vacuum_section_1.CreateEx(TC_Events.Kremer_Events.Takeout_unit_A_error_on_vacuum_section_1, TRUE, 0); 
	Takeout_unit_A_error_on_vacuum_section_2.CreateEx(TC_Events.Kremer_Events.Takeout_unit_A_error_on_vacuum_section_2, TRUE, 0); 
	Takeout_unit_A_error_on_vacuum_section_3.CreateEx(TC_Events.Kremer_Events.Takeout_unit_A_error_on_vacuum_section_3, TRUE, 0); 
	Takeout_unit_A_error_on_vacuum_section_4.CreateEx(TC_Events.Kremer_Events.Takeout_unit_A_error_on_vacuum_section_4, TRUE, 0); 
	Takeout_unit_B_error_on_vacuum_section_1.CreateEx(TC_Events.Kremer_Events.Takeout_unit_B_error_on_vacuum_section_1, TRUE, 0); 
	Takeout_unit_B_error_on_vacuum_section_2.CreateEx(TC_Events.Kremer_Events.Takeout_unit_B_error_on_vacuum_section_2, TRUE, 0); 
	Takeout_unit_B_error_on_vacuum_section_3.CreateEx(TC_Events.Kremer_Events.Takeout_unit_B_error_on_vacuum_section_3, TRUE, 0); 
	Takeout_unit_B_error_on_vacuum_section_4.CreateEx(TC_Events.Kremer_Events.Takeout_unit_B_error_on_vacuum_section_4, TRUE, 0); 
	Machine_pond_hydraulic_pump_maintenance_switch.CreateEx(TC_Events.Kremer_Events.Machine_pond_hydraulic_pump_maintenance_switch, TRUE, 0); 
	Machine_pond_hydraulic_pump_thermal_error.CreateEx(TC_Events.Kremer_Events.Machine_pond_hydraulic_pump_thermal_error, TRUE, 0); 
	Machine_oond_pulp_feeding_cylinder_error.CreateEx(TC_Events.Kremer_Events.Machine_oond_pulp_feeding_cylinder_error, TRUE, 0); 
	Machine_pond_pulp_feeding_cylinder_timeout_in.CreateEx(TC_Events.Kremer_Events.Machine_pond_pulp_feeding_cylinder_timeout_in, TRUE, 0); 
	Machine_pond_pulp_feeding_cylinder_timeout_out.CreateEx(TC_Events.Kremer_Events.Machine_pond_pulp_feeding_cylinder_timeout_out, TRUE, 0); 
	Transfermold_error_on_balluf.CreateEx(TC_Events.Kremer_Events.Transfermold_error_on_balluf, TRUE, 0); 
	Transfermold_is_moving_without_activation.CreateEx(TC_Events.Kremer_Events.Transfermold_is_moving_without_activation, TRUE, 0); 
	RHSR_Bottommold_A_too_cool_for_transfermold_to_come_down.CreateEx(TC_Events.Kremer_Events.RHSR_Bottommold_A_too_cool_for_transfermold_to_come_down, TRUE, 0); 
	RHSR_Bottommold_B_too_cool_for_transfermold_to_come_down.CreateEx(TC_Events.Kremer_Events.RHSR_Bottommold_B_too_cool_for_transfermold_to_come_down, TRUE, 0); 
	Gantry_A_collision_detected.CreateEx(TC_Events.Kremer_Events.Gantry_A_collision_detected, TRUE, 0); 
	Gantry_A_Horizontal_limit_endswitch_backside.CreateEx(TC_Events.Kremer_Events.Gantry_A_Horizontal_limit_endswitch_backside, TRUE, 0); 
	Gantry_A_Horizontal_limit_endswitch_frontside.CreateEx(TC_Events.Kremer_Events.Gantry_A_Horizontal_limit_endswitch_frontside, TRUE, 0); 
	Gantry_A_vertical_limit_endswitch_down.CreateEx(TC_Events.Kremer_Events.Gantry_A_vertical_limit_endswitch_down, TRUE, 0); 
	Gantry_A_vertical_limit_endswitch_up.CreateEx(TC_Events.Kremer_Events.Gantry_A_vertical_limit_endswitch_up, TRUE, 0); 
	Gantry_A_Horizontal_Drive_absoluut_error.CreateEx(TC_Events.Kremer_Events.Gantry_A_Horizontal_Drive_absoluut_error, TRUE, 0); 
	Gantry_A_Horizontal_Drive_Jog_error.CreateEx(TC_Events.Kremer_Events.Gantry_A_Horizontal_Drive_Jog_error, TRUE, 0); 
	Gantry_A_Horizontal_Drive_power_error.CreateEx(TC_Events.Kremer_Events.Gantry_A_Horizontal_Drive_power_error, TRUE, 0); 
	Gantry_A_Horizontal_Drive_reset.CreateEx(TC_Events.Kremer_Events.Gantry_A_Horizontal_Drive_reset, TRUE, 0); 
	Gantry_A_Horizontal_Drive_status.CreateEx(TC_Events.Kremer_Events.Gantry_A_Horizontal_Drive_status, TRUE, 0); 
	Gantry_A_Horizontal_Drive_stop_error.CreateEx(TC_Events.Kremer_Events.Gantry_A_Horizontal_Drive_stop_error, TRUE, 0); 
	Gantry_A_Horizontal_Drive_velocity_error.CreateEx(TC_Events.Kremer_Events.Gantry_A_Horizontal_Drive_velocity_error, TRUE, 0); 
	Gantry_A_Horizontal_Drive_home_error.CreateEx(TC_Events.Kremer_Events.Gantry_A_Horizontal_Drive_home_error, TRUE, 0); 
	Gantry_A_Horizontal_Drive_lag_error.CreateEx(TC_Events.Kremer_Events.Gantry_A_Horizontal_Drive_lag_error, TRUE, 0); 
	Gantry_A_Horizontal_Drive_read_parameter_error.CreateEx(TC_Events.Kremer_Events.Gantry_A_Horizontal_Drive_read_parameter_error, TRUE, 0); 
	Gantry_A_Horizontal_Drive_write_parameter_error.CreateEx(TC_Events.Kremer_Events.Gantry_A_Horizontal_Drive_write_parameter_error, TRUE, 0); 
	Gantry_B_collision_detected.CreateEx(TC_Events.Kremer_Events.Gantry_B_collision_detected, TRUE, 0); 
	Gantry_B_horizontal_limit_endswitch_backside.CreateEx(TC_Events.Kremer_Events.Gantry_B_horizontal_limit_endswitch_backside, TRUE, 0); 
	Gantry_B_horizontal_limit_endswitch_frontside.CreateEx(TC_Events.Kremer_Events.Gantry_B_horizontal_limit_endswitch_frontside, TRUE, 0); 
	Gantry_B_vertical_limit_endswitch_down.CreateEx(TC_Events.Kremer_Events.Gantry_B_vertical_limit_endswitch_down, TRUE, 0); 
	Gantry_B_vertical_limit_endswitch_up.CreateEx(TC_Events.Kremer_Events.Gantry_B_vertical_limit_endswitch_up, TRUE, 0); 
	Gantry_B_Horizontal_Drive_absoluut_error.CreateEx(TC_Events.Kremer_Events.Gantry_B_Horizontal_Drive_absoluut_error, TRUE, 0); 
	Gantry_B_Horizontal_Drive_Jog_error.CreateEx(TC_Events.Kremer_Events.Gantry_B_Horizontal_Drive_Jog_error, TRUE, 0); 
	Gantry_B_Horizontal_Drive_power_error.CreateEx(TC_Events.Kremer_Events.Gantry_B_Horizontal_Drive_power_error, TRUE, 0); 
	Gantry_B_Horizontal_Drive_reset.CreateEx(TC_Events.Kremer_Events.Gantry_B_Horizontal_Drive_reset, TRUE, 0); 
	Gantry_B_Horizontal_Drive_status.CreateEx(TC_Events.Kremer_Events.Gantry_B_Horizontal_Drive_status, TRUE, 0); 
	Gantry_B_Horizontal_Drive_stop_error.CreateEx(TC_Events.Kremer_Events.Gantry_B_Horizontal_Drive_stop_error, TRUE, 0); 
	Gantry_B_Horizontal_Drive_velocity_error.CreateEx(TC_Events.Kremer_Events.Gantry_B_Horizontal_Drive_velocity_error, TRUE, 0); 
	Gantry_B_Horizontal_Drive_home_error.CreateEx(TC_Events.Kremer_Events.Gantry_B_Horizontal_Drive_home_error, TRUE, 0); 
	Gantry_B_Horizontal_Drive_lag_error.CreateEx(TC_Events.Kremer_Events.Gantry_B_Horizontal_Drive_lag_error, TRUE, 0); 
	Gantry_B_Horizontal_Drive_read_parameter_error.CreateEx(TC_Events.Kremer_Events.Gantry_B_Horizontal_Drive_read_parameter_error, TRUE, 0); 
	Gantry_B_Horizontal_Drive_write_parameter_error.CreateEx(TC_Events.Kremer_Events.Gantry_B_Horizontal_Drive_write_parameter_error, TRUE, 0); 
	RHSR_product_handling_gantry_A_is_moving_horizotal_while_vertical_not_on_position.CreateEx(TC_Events.Kremer_Events.RHSR_product_handling_gantry_A_is_moving_horizotal_while_vertical_not_on_position, TRUE, 0); 
	RHSR_product_handling_gantry_B_is_moving_horizotal_while_vertical_not_on_position.CreateEx(TC_Events.Kremer_Events.RHSR_product_handling_gantry_B_is_moving_horizotal_while_vertical_not_on_position, TRUE, 0); 
	RHSR_product_handling_gantry_A_is_moving_vertical_while_horizontal_not_on_position.CreateEx(TC_Events.Kremer_Events.RHSR_product_handling_gantry_A_is_moving_vertical_while_horizontal_not_on_position, TRUE, 0); 
	RHSR_product_handling_gantry_B_is_moving_vertical_while_horizontal_not_on_position.CreateEx(TC_Events.Kremer_Events.RHSR_product_handling_gantry_B_is_moving_vertical_while_horizontal_not_on_position, TRUE, 0); 
	Spraybar_Drive_absoluut_error.CreateEx(TC_Events.Kremer_Events.Spraybar_Drive_absoluut_error, TRUE, 0); 
	Spraybar_Drive_Jog_error.CreateEx(TC_Events.Kremer_Events.Spraybar_Drive_Jog_error, TRUE, 0); 
	Spraybar_Drive_power_error.CreateEx(TC_Events.Kremer_Events.Spraybar_Drive_power_error, TRUE, 0); 
	Spraybar_Drive_reset.CreateEx(TC_Events.Kremer_Events.Spraybar_Drive_reset, TRUE, 0); 
	Spraybar_Drive_status.CreateEx(TC_Events.Kremer_Events.Spraybar_Drive_status, TRUE, 0); 
	Spraybar_Drive_stop_error.CreateEx(TC_Events.Kremer_Events.Spraybar_Drive_stop_error, TRUE, 0); 
	Spraybar_Drive_velocity_error.CreateEx(TC_Events.Kremer_Events.Spraybar_Drive_velocity_error, TRUE, 0); 
	Spraybar_Drive_home_error.CreateEx(TC_Events.Kremer_Events.Spraybar_Drive_home_error, TRUE, 0); 
	Spraybar_Drive_lag_error.CreateEx(TC_Events.Kremer_Events.Spraybar_Drive_lag_error, TRUE, 0); 
	Spraybar_Drive_read_parameter_error.CreateEx(TC_Events.Kremer_Events.Spraybar_Drive_read_parameter_error, TRUE, 0); 
	Spraybar_Drive_write_parameter_error.CreateEx(TC_Events.Kremer_Events.Spraybar_Drive_write_parameter_error, TRUE, 0); 
	Gantry_A_product_lost_section_1.CreateEx(TC_Events.Kremer_Events.Gantry_A_product_lost_section_1, TRUE, 0); 
	Gantry_A_product_lost_section_2.CreateEx(TC_Events.Kremer_Events.Gantry_A_product_lost_section_2, TRUE, 0); 
	Gantry_A_product_lost_section_3.CreateEx(TC_Events.Kremer_Events.Gantry_A_product_lost_section_3, TRUE, 0); 
	Gantry_A_product_lost_section_4.CreateEx(TC_Events.Kremer_Events.Gantry_A_product_lost_section_4, TRUE, 0); 
	Gantry_A_product_lost_section_5.CreateEx(TC_Events.Kremer_Events.Gantry_A_product_lost_section_5, TRUE, 0); 
	Gantry_A_product_lost_section_6.CreateEx(TC_Events.Kremer_Events.Gantry_A_product_lost_section_6, TRUE, 0); 
	Gantry_B_product_lost_section_1.CreateEx(TC_Events.Kremer_Events.Gantry_B_product_lost_section_1, TRUE, 0); 
	Gantry_B_product_lost_section_2.CreateEx(TC_Events.Kremer_Events.Gantry_B_product_lost_section_2, TRUE, 0); 
	Gantry_B_product_lost_section_3.CreateEx(TC_Events.Kremer_Events.Gantry_B_product_lost_section_3, TRUE, 0); 
	Gantry_B_product_lost_section_4.CreateEx(TC_Events.Kremer_Events.Gantry_B_product_lost_section_4, TRUE, 0); 
	Gantry_B_product_lost_section_5.CreateEx(TC_Events.Kremer_Events.Gantry_B_product_lost_section_5, TRUE, 0); 
	Gantry_B_product_lost_section_6.CreateEx(TC_Events.Kremer_Events.Gantry_B_product_lost_section_6, TRUE, 0); 
	Spraybar_not_in_front_rest_position.CreateEx(TC_Events.Kremer_Events.Spraybar_not_in_front_rest_position, TRUE, 0); 
	Spraybar_not_in_back_rest_position.CreateEx(TC_Events.Kremer_Events.Spraybar_not_in_back_rest_position, TRUE, 0); 
	Ethercat_diagnosed_a_link_error.CreateEx(TC_Events.Kremer_Events.Ethercat_diagnosed_a_link_error, TRUE, 0); 
	Ethercat_diagnosed_that_a_slave_is_missing.CreateEx(TC_Events.Kremer_Events.Ethercat_diagnosed_that_a_slave_is_missing, TRUE, 0); 
	Ethercat_diagnosed_a_non_OP_state.CreateEx(TC_Events.Kremer_Events.Ethercat_diagnosed_a_non_OP_state, TRUE, 0); 
	Ethercat_diagnosed_that_a_ethercat_reset_is_needed.CreateEx(TC_Events.Kremer_Events.Ethercat_diagnosed_that_a_ethercat_reset_is_needed, TRUE, 0); 
	TopMold_A_Safe_position_not_reached.CreateEx(TC_Events.Kremer_Events.TopMold_A_Safe_position_not_reached, TRUE, 0); 
	TopMold_B_Safe_position_not_reached.CreateEx(TC_Events.Kremer_Events.TopMold_B_Safe_position_not_reached, TRUE, 0); 
	Transfermold_Safe_position_not_reached.CreateEx(TC_Events.Kremer_Events.Transfermold_Safe_position_not_reached, TRUE, 0); 
	Difference_in_temperature_too_high_top_bottommold_A_zone_1.CreateEx(TC_Events.Kremer_Events.Difference_in_temperature_too_high_top_bottommold_A_zone_1, TRUE, 0); 
	Difference_in_temperature_too_high_top_bottommold_A_zone_2.CreateEx(TC_Events.Kremer_Events.Difference_in_temperature_too_high_top_bottommold_A_zone_2, TRUE, 0); 
	Difference_in_temperature_too_high_top_bottommold_A_zone_3.CreateEx(TC_Events.Kremer_Events.Difference_in_temperature_too_high_top_bottommold_A_zone_3, TRUE, 0); 
	Difference_in_temperature_too_high_top_bottommold_A_zone_4.CreateEx(TC_Events.Kremer_Events.Difference_in_temperature_too_high_top_bottommold_A_zone_4, TRUE, 0); 
	Difference_in_temperature_too_high_top_bottommold_A_zone_5.CreateEx(TC_Events.Kremer_Events.Difference_in_temperature_too_high_top_bottommold_A_zone_5, TRUE, 0); 
	Difference_in_temperature_too_high_top_bottommold_A_zone_6.CreateEx(TC_Events.Kremer_Events.Difference_in_temperature_too_high_top_bottommold_A_zone_6, TRUE, 0); 
	Difference_in_temperature_too_high_top_bottommold_B_zone_1.CreateEx(TC_Events.Kremer_Events.Difference_in_temperature_too_high_top_bottommold_B_zone_1, TRUE, 0); 
	Difference_in_temperature_too_high_top_bottommold_B_zone_2.CreateEx(TC_Events.Kremer_Events.Difference_in_temperature_too_high_top_bottommold_B_zone_2, TRUE, 0); 
	Difference_in_temperature_too_high_top_bottommold_B_zone_3.CreateEx(TC_Events.Kremer_Events.Difference_in_temperature_too_high_top_bottommold_B_zone_3, TRUE, 0); 
	Difference_in_temperature_too_high_top_bottommold_B_zone_4.CreateEx(TC_Events.Kremer_Events.Difference_in_temperature_too_high_top_bottommold_B_zone_4, TRUE, 0); 
	Difference_in_temperature_too_high_top_bottommold_B_zone_5.CreateEx(TC_Events.Kremer_Events.Difference_in_temperature_too_high_top_bottommold_B_zone_5, TRUE, 0); 
	Difference_in_temperature_too_high_top_bottommold_B_zone_6.CreateEx(TC_Events.Kremer_Events.Difference_in_temperature_too_high_top_bottommold_B_zone_6, TRUE, 0); 
	Gantry_A_Vertical_Drive_absoluut_error.CreateEx(TC_Events.Kremer_Events.Gantry_A_Vertical_Drive_absoluut_error, TRUE, 0); 
	Gantry_A_Vertical_Drive_Jog_error.CreateEx(TC_Events.Kremer_Events.Gantry_A_Vertical_Drive_Jog_error, TRUE, 0); 
	Gantry_A_Vertical_Drive_power_error.CreateEx(TC_Events.Kremer_Events.Gantry_A_Vertical_Drive_power_error, TRUE, 0); 
	Gantry_A_Vertical_Drive_reset.CreateEx(TC_Events.Kremer_Events.Gantry_A_Vertical_Drive_reset, TRUE, 0); 
	Gantry_A_Vertical_Drive_status.CreateEx(TC_Events.Kremer_Events.Gantry_A_Vertical_Drive_status, TRUE, 0); 
	Gantry_A_Vertical_Drive_stop_error.CreateEx(TC_Events.Kremer_Events.Gantry_A_Vertical_Drive_stop_error, TRUE, 0); 
	Gantry_A_Vertical_Drive_velocity_error.CreateEx(TC_Events.Kremer_Events.Gantry_A_Vertical_Drive_velocity_error, TRUE, 0); 
	Gantry_A_Vertical_Drive_home_error.CreateEx(TC_Events.Kremer_Events.Gantry_A_Vertical_Drive_home_error, TRUE, 0); 
	Gantry_A_Vertical_Drive_lag_error.CreateEx(TC_Events.Kremer_Events.Gantry_A_Vertical_Drive_lag_error, TRUE, 0); 
	Gantry_A_Vertical_Drive_read_parameter_error.CreateEx(TC_Events.Kremer_Events.Gantry_A_Vertical_Drive_read_parameter_error, TRUE, 0); 
	Gantry_A_Vertical_Drive_write_parameter_error.CreateEx(TC_Events.Kremer_Events.Gantry_A_Vertical_Drive_write_parameter_error, TRUE, 0); 
	Gantry_B_Vertical_Drive_absoluut_error.CreateEx(TC_Events.Kremer_Events.Gantry_B_Vertical_Drive_absoluut_error, TRUE, 0); 
	Gantry_B_Vertical_Drive_Jog_error.CreateEx(TC_Events.Kremer_Events.Gantry_B_Vertical_Drive_Jog_error, TRUE, 0); 
	Gantry_B_Vertical_Drive_power_error.CreateEx(TC_Events.Kremer_Events.Gantry_B_Vertical_Drive_power_error, TRUE, 0); 
	Gantry_B_Vertical_Drive_reset.CreateEx(TC_Events.Kremer_Events.Gantry_B_Vertical_Drive_reset, TRUE, 0); 
	Gantry_B_Vertical_Drive_status.CreateEx(TC_Events.Kremer_Events.Gantry_B_Vertical_Drive_status, TRUE, 0); 
	Gantry_B_Vertical_Drive_stop_error.CreateEx(TC_Events.Kremer_Events.Gantry_B_Vertical_Drive_stop_error, TRUE, 0); 
	Gantry_B_Vertical_Drive_velocity_error.CreateEx(TC_Events.Kremer_Events.Gantry_B_Vertical_Drive_velocity_error, TRUE, 0); 
	Gantry_B_Vertical_Drive_home_error.CreateEx(TC_Events.Kremer_Events.Gantry_B_Vertical_Drive_home_error, TRUE, 0); 
	Gantry_B_Vertical_Drive_lag_error.CreateEx(TC_Events.Kremer_Events.Gantry_B_Vertical_Drive_lag_error, TRUE, 0); 
	Gantry_B_Vertical_Drive_read_parameter_error.CreateEx(TC_Events.Kremer_Events.Gantry_B_Vertical_Drive_read_parameter_error, TRUE, 0); 
	Gantry_B_Vertical_Drive_write_parameter_error.CreateEx(TC_Events.Kremer_Events.Gantry_B_Vertical_Drive_write_parameter_error, TRUE, 0); 
	Bottommold_B_Horizontal_Drive_absoluut_error.CreateEx(TC_Events.Kremer_Events.Bottommold_B_Horizontal_Drive_absoluut_error, TRUE, 0); 
	Bottommold_B_Horizontal_Drive_Jog_error.CreateEx(TC_Events.Kremer_Events.Bottommold_B_Horizontal_Drive_Jog_error, TRUE, 0); 
	Bottommold_B_Horizontal_Drive_power_error.CreateEx(TC_Events.Kremer_Events.Bottommold_B_Horizontal_Drive_power_error, TRUE, 0); 
	Bottommold_B_Horizontal_Drive_reset.CreateEx(TC_Events.Kremer_Events.Bottommold_B_Horizontal_Drive_reset, TRUE, 0); 
	Bottommold_B_Horizontal_Drive_status.CreateEx(TC_Events.Kremer_Events.Bottommold_B_Horizontal_Drive_status, TRUE, 0); 
	Bottommold_B_Horizontal_Drive_stop_error.CreateEx(TC_Events.Kremer_Events.Bottommold_B_Horizontal_Drive_stop_error, TRUE, 0); 
	Bottommold_B_Horizontal_Drive_velocity_error.CreateEx(TC_Events.Kremer_Events.Bottommold_B_Horizontal_Drive_velocity_error, TRUE, 0); 
	Bottommold_B_Horizontal_Drive_home_error.CreateEx(TC_Events.Kremer_Events.Bottommold_B_Horizontal_Drive_home_error, TRUE, 0); 
	Bottommold_B_Horizontal_Drive_lag_error.CreateEx(TC_Events.Kremer_Events.Bottommold_B_Horizontal_Drive_lag_error, TRUE, 0); 
	Bottommold_B_Horizontal_Drive_read_parameter_error.CreateEx(TC_Events.Kremer_Events.Bottommold_B_Horizontal_Drive_read_parameter_error, TRUE, 0); 
	Bottommold_B_Horizontal_Drive_write_parameter_error.CreateEx(TC_Events.Kremer_Events.Bottommold_B_Horizontal_Drive_write_parameter_error, TRUE, 0); 
	Bottommold_A_Horizontal_Drive_absoluut_error.CreateEx(TC_Events.Kremer_Events.Bottommold_A_Horizontal_Drive_absoluut_error, TRUE, 0); 
	Bottommold_A_Horizontal_Drive_Jog_error.CreateEx(TC_Events.Kremer_Events.Bottommold_A_Horizontal_Drive_Jog_error, TRUE, 0); 
	Bottommold_A_Horizontal_Drive_power_error.CreateEx(TC_Events.Kremer_Events.Bottommold_A_Horizontal_Drive_power_error, TRUE, 0); 
	Bottommold_A_Horizontal_Drive_reset.CreateEx(TC_Events.Kremer_Events.Bottommold_A_Horizontal_Drive_reset, TRUE, 0); 
	Bottommold_A_Horizontal_Drive_status.CreateEx(TC_Events.Kremer_Events.Bottommold_A_Horizontal_Drive_status, TRUE, 0); 
	Bottommold_A_Horizontal_Drive_stop_error.CreateEx(TC_Events.Kremer_Events.Bottommold_A_Horizontal_Drive_stop_error, TRUE, 0); 
	Bottommold_A_Horizontal_Drive_velocity_error.CreateEx(TC_Events.Kremer_Events.Bottommold_A_Horizontal_Drive_velocity_error, TRUE, 0); 
	Bottommold_A_Horizontal_Drive_home_error.CreateEx(TC_Events.Kremer_Events.Bottommold_A_Horizontal_Drive_home_error, TRUE, 0); 
	Bottommold_A_Horizontal_Drive_lag_error.CreateEx(TC_Events.Kremer_Events.Bottommold_A_Horizontal_Drive_lag_error, TRUE, 0); 
	Bottommold_A_Horizontal_Drive_read_parameter_error.CreateEx(TC_Events.Kremer_Events.Bottommold_A_Horizontal_Drive_read_parameter_error, TRUE, 0); 
	Bottommold_A_Horizontal_Drive_write_parameter_error.CreateEx(TC_Events.Kremer_Events.Bottommold_A_Horizontal_Drive_write_parameter_error, TRUE, 0); 
END_IF 

IF Main.Errors.exEmergency[1] THEN 
Emergency_zone_1.Raise(0); 
END_IF 

IF Main.Errors.exEmergency[2] THEN 
Emergency_zone_2.Raise(0); 
END_IF 

IF Main.Errors.exEmergency[3] THEN 
Emergency_zone_3.Raise(0); 
END_IF 

IF Main.Errors.exEmergency[4] THEN 
Emergency_zone_4.Raise(0); 
END_IF 

IF Main.Errors.exEmergency[5] THEN 
Emergency_zone_5.Raise(0); 
END_IF 

IF Main.Errors.exEmergency[6] THEN 
Emergency_zone_6.Raise(0); 
END_IF 

IF Main.Errors.exEmergency[7] THEN 
Emergency_zone_7.Raise(0); 
END_IF 

IF Main.Errors.exEmStopImdFront THEN 
In_mold_drying_emergency_stop_pressed_front_side.Raise(0); 
END_IF 

IF Main.Errors.exEmStopImdBack THEN 
In_mold_drying_emergency_stop_pressed_back_side.Raise(0); 
END_IF 

IF Main.Errors.exImdFrontDoorLeft THEN 
In_mold_drying_door_opend_frontside_left.Raise(0); 
END_IF 

IF Main.Errors.exImdFrontDoorMiddle THEN 
In_mold_drying_door_opened_frontside_middle.Raise(0); 
END_IF 

IF Main.Errors.exImdFrontDoorRight THEN 
In_mold_drying_door_opened_frontside_right.Raise(0); 
END_IF 

IF Main.Errors.exImdBackDoorLeft1 THEN 
In_mold_drying_double_door_opened_backside_left_1.Raise(0); 
END_IF 

IF Main.Errors.exImdBackDoorLeft2 THEN 
In_mold_drying_double_door_opened_backside_left_2.Raise(0); 
END_IF 

IF Main.Errors.exImdBackDoorMiddle3 THEN 
In_mold_drying_double_door_opened_backside_Middle_1.Raise(0); 
END_IF 

IF Main.Errors.exImdBackDoorMiddle4 THEN 
In_mold_drying_double_door_opened_backside_Middle_2.Raise(0); 
END_IF 

IF Main.Errors.exImdBackDoorRight5 THEN 
In_mold_drying_double_door_opened_backside_Right_1.Raise(0); 
END_IF 

IF Main.Errors.exImdBackDoorRight6 THEN 
In_mold_drying_double_door_opened_backside_Right_2.Raise(0); 
END_IF 

IF Main.Errors.exGantryA_FrontDoorLeft THEN 
Gantry_A_front_door_openend_right.Raise(0); 
END_IF 

IF Main.Errors.exGantryA_FrontDoorRight THEN 
Gantry_A_front_door_openend_left.Raise(0); 
END_IF 

IF Main.Errors.exGantryA_BackDoor THEN 
Gantry_A_Back_door_openend.Raise(0); 
END_IF 

IF Main.Errors.exGantryB_FrontDoorLeft THEN 
Gantry_B_front_door_openend_left.Raise(0); 
END_IF 

IF Main.Errors.exGantryB_FrontDoorRight THEN 
Gantry_B_front_door_openend_right.Raise(0); 
END_IF 

IF Main.Errors.exGantryB_BackDoor THEN 
Gantry_B_Back_door_openend.Raise(0); 
END_IF 

IF Main.Errors.exEmStopGantryA_Back THEN 
Emergency_stop_pressed_Gantry_A_backside.Raise(0); 
END_IF 

IF Main.Errors.exEmStopGantryA_Front THEN 
Emergency_stop_pressed_Gantry_A_Frontside.Raise(0); 
END_IF 

IF Main.Errors.exEmStopGantryB_Back THEN 
Emergency_stop_pressed_Gantry_B_Backside.Raise(0); 
END_IF 

IF Main.Errors.exEmStopGantryB_Front THEN 
Emergency_stop_pressed_Gantry_B_Frontside.Raise(0); 
END_IF 

IF Main.Errors.ex24VoltError1 THEN 
_24_volt_circuit_in_error_1.Raise(0); 
END_IF 

IF Main.Errors.ex24VoltError2 THEN 
_24_volt_circuit_in_error_2.Raise(0); 
END_IF 

IF Main.Errors.exAtteptedStartWithNoProduct THEN 
No_product_loaded_please_load_a_valid_product_first.Raise(0); 
END_IF 

IF Main.Errors.MainAirSupplyError THEN 
Main_air_supply_has_an_error.Raise(0); 
END_IF 

IF Main.InMoldDrying.Errors.HydraulicMain.HydraulicPump.SofstarterFailure THEN 
In_mold_drying_hydraulic_pump_softstarter_failure.Raise(0); 
END_IF 

IF Main.InMoldDrying.Errors.HydraulicMain.HydraulicPump.Maintenance THEN 
In_mold_drying_hydraulic_pump_maintenance_switch.Raise(0); 
END_IF 

IF Main.InMoldDrying.Errors.HydraulicMain.Coolingfan.Thermal THEN 
In_mold_drying_cooling_fan_thermal_failure.Raise(0); 
END_IF 

IF Main.InMoldDrying.Errors.HydraulicMain.Coolingfan.Maintenance THEN 
In_mold_drying_cooling_fan_maintenance_switch.Raise(0); 
END_IF 

IF Main.InMoldDrying.Errors.HydraulicMain.FilterMotor.Thermal THEN 
In_mold_drying_filter_motor_thermal.Raise(0); 
END_IF 

IF Main.InMoldDrying.Errors.HydraulicMain.FilterMotor.Maintenance THEN 
In_mold_drying_filter_motor_maintenance.Raise(0); 
END_IF 

IF Main.InMoldDrying.Errors.ProductForming.CssHasError THEN 
Css_has_an_active_error.Raise(0); 
END_IF 

IF Main.InMoldDrying.Errors.ProductForming.LowLvlOnBothTanks THEN 
Both_Pulp_Tanks_below_Low_Level_stopping_IMD.Raise(0); 
END_IF 

IF Main.InMoldDrying.Errors.RH_BoMoldAIsMovingToMoldANotInPos THEN 
RHSR_Bottom_mold_A_moving_while_top_mold_A_not_in_position.Raise(0); 
END_IF 

IF Main.InMoldDrying.Errors.RH_BoMoldAIsMovingTrMoldNotInPos THEN 
RHSR_Bottom_mold_A_moving_while_transfer_mold_A_not_in_position.Raise(0); 
END_IF 

IF Main.InMoldDrying.Errors.RH_BoMoldBIsMovingToMoldBNotInPos THEN 
RHSR_Bottom_mold_B_moving_while_top_mold_B_not_in_position.Raise(0); 
END_IF 

IF Main.InMoldDrying.Errors.RH_BoMoldBIsMovingTrMoldNotInPos THEN 
RHSR_Bottom_mold_B_moving_while_transfer_mold_B_not_in_position.Raise(0); 
END_IF 

IF Main.InMoldDrying.Errors.RH_TaOutHorAIsMovingVertIsNotDown THEN 
RHSR_Takeout_A_moving_while_vertical_cylinder_is_not_down.Raise(0); 
END_IF 

IF Main.InMoldDrying.Errors.RH_TaOutHorBIsMovingVertIsNotDown THEN 
RHSR_Takeout_B_moving_while_vertical_cylinder_is_not_down.Raise(0); 
END_IF 

IF Main.InMoldDrying.Errors.RH_ToMoldAIsMovingBoMoldANotInPos THEN 
RHSR_TopMold_A_moving_while_bottom_mold_A_is_not_in_position.Raise(0); 
END_IF 

IF Main.InMoldDrying.Errors.RH_ToMoldBIsMovingBoMoldBNotInPos THEN 
RHSR_TopMold_B_moving_while_bottom_mold_B_is_not_in_position.Raise(0); 
END_IF 

IF Main.InMoldDrying.Errors.RH_TrMoldIsMovingBoMoldANotInPos THEN 
RHSR_Transfermold_moving_while_bottom_mold_A_is_not_in_posititon.Raise(0); 
END_IF 

IF Main.InMoldDrying.Errors.RH_TrMoldIsMovingBoMoldBNotInPos THEN 
RHSR_Transfermold_moving_while_bottom_mold_B_is_not_in_position.Raise(0); 
END_IF 

IF Main.InMoldDrying.Errors.RH_TrMoldIsMovingSprayBNotInPos THEN 
RHSR_Transfermold_moving_while_spraybar_is_not_at_one_of_rest_positions.Raise(0); 
END_IF 

IF Main.InMoldDrying.Errors.TempDiffTopBottomTooHigh_SideA THEN 
Temperature_difference_between_top_and_bottom_mold_side_A_to_high.Raise(0); 
END_IF 

IF Main.InMoldDrying.Errors.TempDiffTopBottomTooHigh_SideB THEN 
Temperature_difference_between_top_and_bottom_mold_side_B_to_high.Raise(0); 
END_IF 

IF Main.InMoldDrying.Errors.RH_SprayBIsMovingTrNotClear THEN 
Spare56.Raise(0); 
END_IF 

IF Main.InMoldDrying.Errors.HydraulicMain.AuxFilter100Dirty THEN 
Auxiliary_filter_100_dirty.Raise(0); 
END_IF 

IF Main.InMoldDrying.Errors.HydraulicMain.AuxFilter75Dirty THEN 
Auxiliary_filter_75_dirty.Raise(0); 
END_IF 

IF Main.InMoldDrying.Errors.HydraulicMain.Filter100Dirty THEN 
Oil_filter_100_dirty.Raise(0); 
END_IF 

IF Main.InMoldDrying.Errors.HydraulicMain.Filter75Dirty THEN 
Oil_filter_75_dirty.Raise(0); 
END_IF 

IF Main.InMoldDrying.Errors.HydraulicMain.CoolingFanCabinet THEN 
Fan_on_MCC2_error.Raise(0); 
END_IF 

IF Main.InMoldDrying.Errors.HydraulicMain.Hydraulics24VError THEN 
_24V_error_on_MCC2.Raise(0); 
END_IF 

IF Main.InMoldDrying.Errors.HydraulicMain.OilLevelTooLow THEN 
Oil_temperature_too_low.Raise(0); 
END_IF 

IF Main.InMoldDrying.Errors.HydraulicMain.OilTemperatureTooHigh THEN 
Oil_temperature_too_high.Raise(0); 
END_IF 

IF Main.Errors.InMoldDryingErrors.TopMoldA.Hydraulic.BallufError THEN 
Top_mold_A_error_on_balluf.Raise(0); 
END_IF 

IF Main.Errors.InMoldDryingErrors.TopMoldA.TmDidNotReachBmPosTimeOut							 THEN 
Top_mold_A_position_error.Raise(0); 
END_IF 

IF Main.Errors.InMoldDryingErrors.TopMoldA.Hydraulic.IsMovingWithoutActivation THEN 
Top_mold_A_timed_out_Did_not_reach_bottommold_position_in_time.Raise(0); 
END_IF 

IF FALSE THEN 
Top_mold_A_Rod_side_pressure_too_high.Raise(0); 
END_IF 

IF FALSE THEN 
Top_mold_A_Bot_side_pressure_too_high.Raise(0); 
END_IF 

IF Main.Errors.InMoldDryingErrors.TopMoldA.HeatingZone[1].PT100_ConnectorNotConnected THEN 
Topmold_A_heating_zone_1_connector_not_connected.Raise(0); 
END_IF 

IF Main.Errors.InMoldDryingErrors.TopMoldA.HeatingZone[1].PT100_HasWrongPosition THEN 
Topmold_A_heating_zone_1_PT100_wrong_position.Raise(0); 
END_IF 

IF Main.Errors.InMoldDryingErrors.TopMoldA.HeatingZone[1].PT100_Loose THEN 
Topmold_A_heating_zone_1_PT100_loose.Raise(0); 
END_IF 

IF Main.Errors.InMoldDryingErrors.TopMoldA.HeatingZone[1].PT100_NotInserted THEN 
Topmold_A_heating_zone_1_PT100_not_inserted.Raise(0); 
END_IF 

IF Main.Errors.InMoldDryingErrors.TopMoldA.HeatingZone[1].PT100_TempAboveSetpoint THEN 
Topmold_A_heating_zone_1_Temperature_above_setpoint.Raise(0); 
END_IF 

IF Main.Errors.InMoldDryingErrors.TopMoldA.HeatingZone[1].PT100_TempBelowSetpoint THEN 
Topmold_A_heating_zone_1_Temperature_below_setpoint.Raise(0); 
END_IF 

IF Main.Errors.InMoldDryingErrors.TopMoldA.HeatingZone[1].PT100_WireBreak THEN 
Topmold_A_heating_zone_1_PT100_wirebreak.Raise(0); 
END_IF 

IF Main.Errors.InMoldDryingErrors.TopMoldA.HeatingZone[1].Thermal THEN 
Topmold_A_heating_zone_1_Thermal.Raise(0); 
END_IF 

IF Main.Errors.InMoldDryingErrors.TopMoldA.HeatingZone[1].PT100_TemperatureAboveMaximum THEN 
Topmold_A_heating_zone_1_temperature_above_250_degree_heating_element_switched_off.Raise(0); 
END_IF 

IF Main.Errors.InMoldDryingErrors.TopMoldA.HeatingZone[1].PT100_TemperatureTooHighWarn THEN 
Topmold_A_heating_zone_1_temperature_above_230_degree.Raise(0); 
END_IF 

IF Main.Errors.InMoldDryingErrors.TopMoldA.HeatingZone[2].PT100_ConnectorNotConnected THEN 
Topmold_A_heating_zone_2_connector_not_connected.Raise(0); 
END_IF 

IF Main.Errors.InMoldDryingErrors.TopMoldA.HeatingZone[2].PT100_HasWrongPosition THEN 
Topmold_A_heating_zone_2_PT100_wrong_position.Raise(0); 
END_IF 

IF Main.Errors.InMoldDryingErrors.TopMoldA.HeatingZone[2].PT100_Loose THEN 
Topmold_A_heating_zone_2_PT100_loose.Raise(0); 
END_IF 

IF Main.Errors.InMoldDryingErrors.TopMoldA.HeatingZone[2].PT100_NotInserted THEN 
Topmold_A_heating_zone_2_PT100_not_inserted.Raise(0); 
END_IF 

IF Main.Errors.InMoldDryingErrors.TopMoldA.HeatingZone[2].PT100_TempAboveSetpoint THEN 
Topmold_A_heating_zone_2_Temperature_above_setpoint.Raise(0); 
END_IF 

IF Main.Errors.InMoldDryingErrors.TopMoldA.HeatingZone[2].PT100_TempBelowSetpoint THEN 
Topmold_A_heating_zone_2_Temperature_below_setpoint.Raise(0); 
END_IF 

IF Main.Errors.InMoldDryingErrors.TopMoldA.HeatingZone[2].PT100_WireBreak THEN 
Topmold_A_heating_zone_2_PT100_wirebreak.Raise(0); 
END_IF 

IF Main.Errors.InMoldDryingErrors.TopMoldA.HeatingZone[2].Thermal THEN 
Topmold_A_heating_zone_2_Thermal.Raise(0); 
END_IF 

IF Main.Errors.InMoldDryingErrors.TopMoldA.HeatingZone[2].PT100_TemperatureAboveMaximum THEN 
Topmold_A_heating_zone_2_temperature_above_250_degree_heating_element_switched_off.Raise(0); 
END_IF 

IF Main.Errors.InMoldDryingErrors.TopMoldA.HeatingZone[2].PT100_TemperatureTooHighWarn THEN 
Topmold_A_heating_zone_2_temperature_above_230_degree.Raise(0); 
END_IF 

IF Main.Errors.InMoldDryingErrors.TransferMold.TrDidNotReachBMPosTimeOut							 THEN 
Tranfermold_timed_out_did_not_reach_bottommold_position_in_time.Raise(0); 
END_IF 

IF Main.Errors.InMoldDryingErrors.TransferMold.TrDidNotReachFormingPosTimeOut	 THEN 
Tranfermold_timed_out_did_not_reach_forming_position_in_time.Raise(0); 
END_IF 

IF Main.Errors.InMoldDryingErrors.TopMoldA.HeatingZone[3].PT100_ConnectorNotConnected THEN 
Topmold_A_heating_zone_3_connector_not_connected.Raise(0); 
END_IF 

IF Main.Errors.InMoldDryingErrors.TopMoldA.HeatingZone[3].PT100_HasWrongPosition THEN 
Topmold_A_heating_zone_3_PT100_wrong_position.Raise(0); 
END_IF 

IF Main.Errors.InMoldDryingErrors.TopMoldA.HeatingZone[3].PT100_Loose THEN 
Topmold_A_heating_zone_3_PT100_loose.Raise(0); 
END_IF 

IF Main.Errors.InMoldDryingErrors.TopMoldA.HeatingZone[3].PT100_NotInserted THEN 
Topmold_A_heating_zone_3_PT100_not_inserted.Raise(0); 
END_IF 

IF Main.Errors.InMoldDryingErrors.TopMoldA.HeatingZone[3].PT100_TempAboveSetpoint THEN 
Topmold_A_heating_zone_3_Temperature_above_setpoint.Raise(0); 
END_IF 

IF Main.Errors.InMoldDryingErrors.TopMoldA.HeatingZone[3].PT100_TempBelowSetpoint THEN 
Topmold_A_heating_zone_3_Temperature_below_setpoint.Raise(0); 
END_IF 

IF Main.Errors.InMoldDryingErrors.TopMoldA.HeatingZone[3].PT100_WireBreak THEN 
Topmold_A_heating_zone_3_PT100_wirebreak.Raise(0); 
END_IF 

IF Main.Errors.InMoldDryingErrors.TopMoldA.HeatingZone[3].Thermal THEN 
Topmold_A_heating_zone_3_Thermal.Raise(0); 
END_IF 

IF Main.Errors.InMoldDryingErrors.TopMoldA.HeatingZone[3].PT100_TemperatureAboveMaximum THEN 
Topmold_A_heating_zone_3_temperature_above_250_degree_heating_element_switched_off.Raise(0); 
END_IF 

IF Main.Errors.InMoldDryingErrors.TopMoldA.HeatingZone[3].PT100_TemperatureTooHighWarn THEN 
Topmold_A_heating_zone_3_temperature_above_230_degree.Raise(0); 
END_IF 

IF Main.Errors.InMoldDryingErrors.TopMoldA.HeatingZone[4].PT100_ConnectorNotConnected THEN 
Topmold_A_heating_zone_4_connector_not_connected.Raise(0); 
END_IF 

IF Main.Errors.InMoldDryingErrors.TopMoldA.HeatingZone[4].PT100_HasWrongPosition THEN 
Topmold_A_heating_zone_4_PT100_wrong_position.Raise(0); 
END_IF 

IF Main.Errors.InMoldDryingErrors.TopMoldA.HeatingZone[4].PT100_Loose THEN 
Topmold_A_heating_zone_4_PT100_loose.Raise(0); 
END_IF 

IF Main.Errors.InMoldDryingErrors.TopMoldA.HeatingZone[4].PT100_NotInserted THEN 
Topmold_A_heating_zone_4_PT100_not_inserted.Raise(0); 
END_IF 

IF Main.Errors.InMoldDryingErrors.TopMoldA.HeatingZone[4].PT100_TempAboveSetpoint THEN 
Topmold_A_heating_zone_4_Temperature_above_setpoint.Raise(0); 
END_IF 

IF Main.Errors.InMoldDryingErrors.TopMoldA.HeatingZone[4].PT100_TempBelowSetpoint THEN 
Topmold_A_heating_zone_4_Temperature_below_setpoint.Raise(0); 
END_IF 

IF Main.Errors.InMoldDryingErrors.TopMoldA.HeatingZone[4].PT100_WireBreak THEN 
Topmold_A_heating_zone_4_PT100_wirebreak.Raise(0); 
END_IF 

IF Main.Errors.InMoldDryingErrors.TopMoldA.HeatingZone[4].Thermal THEN 
Topmold_A_heating_zone_4_Thermal.Raise(0); 
END_IF 

IF Main.Errors.InMoldDryingErrors.TopMoldA.HeatingZone[4].PT100_TemperatureAboveMaximum THEN 
Topmold_A_heating_zone_4_temperature_above_250_degree_heating_element_switched_off.Raise(0); 
END_IF 

IF Main.Errors.InMoldDryingErrors.TopMoldA.HeatingZone[4].PT100_TemperatureTooHighWarn THEN 
Topmold_A_heating_zone_4_temperature_above_230_degree.Raise(0); 
END_IF 

IF Main.Errors.InMoldDryingErrors.TopMoldA.HeatingZone[5].PT100_ConnectorNotConnected THEN 
Topmold_A_heating_zone_5_connector_not_connected.Raise(0); 
END_IF 

IF Main.Errors.InMoldDryingErrors.TopMoldA.HeatingZone[5].PT100_HasWrongPosition THEN 
Topmold_A_heating_zone_5_PT100_wrong_position.Raise(0); 
END_IF 

IF Main.Errors.InMoldDryingErrors.TopMoldA.HeatingZone[5].PT100_Loose THEN 
Topmold_A_heating_zone_5_PT100_loose.Raise(0); 
END_IF 

IF Main.Errors.InMoldDryingErrors.TopMoldA.HeatingZone[5].PT100_NotInserted THEN 
Topmold_A_heating_zone_5_PT100_not_inserted.Raise(0); 
END_IF 

IF Main.Errors.InMoldDryingErrors.TopMoldA.HeatingZone[5].PT100_TempAboveSetpoint THEN 
Topmold_A_heating_zone_5_Temperature_above_setpoint.Raise(0); 
END_IF 

IF Main.Errors.InMoldDryingErrors.TopMoldA.HeatingZone[5].PT100_TempBelowSetpoint THEN 
Topmold_A_heating_zone_5_Temperature_below_setpoint.Raise(0); 
END_IF 

IF Main.Errors.InMoldDryingErrors.TopMoldA.HeatingZone[5].PT100_WireBreak THEN 
Topmold_A_heating_zone_5_PT100_wirebreak.Raise(0); 
END_IF 

IF Main.Errors.InMoldDryingErrors.TopMoldA.HeatingZone[5].Thermal THEN 
Topmold_A_heating_zone_5_Thermal.Raise(0); 
END_IF 

IF Main.Errors.InMoldDryingErrors.TopMoldA.HeatingZone[5].PT100_TemperatureAboveMaximum THEN 
Topmold_A_heating_zone_5_temperature_above_250_degree_heating_element_switched_off.Raise(0); 
END_IF 

IF Main.Errors.InMoldDryingErrors.TopMoldA.HeatingZone[5].PT100_TemperatureTooHighWarn THEN 
Topmold_A_heating_zone_5_temperature_above_230_degree.Raise(0); 
END_IF 

IF Main.Errors.InMoldDryingErrors.TopMoldA.HeatingZone[6].PT100_ConnectorNotConnected THEN 
Topmold_A_heating_zone_6_connector_not_connected.Raise(0); 
END_IF 

IF Main.Errors.InMoldDryingErrors.TopMoldA.HeatingZone[6].PT100_HasWrongPosition THEN 
Topmold_A_heating_zone_6_PT100_wrong_position.Raise(0); 
END_IF 

IF Main.Errors.InMoldDryingErrors.TopMoldA.HeatingZone[6].PT100_Loose THEN 
Topmold_A_heating_zone_6_PT100_loose.Raise(0); 
END_IF 

IF Main.Errors.InMoldDryingErrors.TopMoldA.HeatingZone[6].PT100_NotInserted THEN 
Topmold_A_heating_zone_6_PT100_not_inserted.Raise(0); 
END_IF 

IF Main.Errors.InMoldDryingErrors.TopMoldA.HeatingZone[6].PT100_TempAboveSetpoint THEN 
Topmold_A_heating_zone_6_Temperature_above_setpoint.Raise(0); 
END_IF 

IF Main.Errors.InMoldDryingErrors.TopMoldA.HeatingZone[6].PT100_TempBelowSetpoint THEN 
Topmold_A_heating_zone_6_Temperature_below_setpoint.Raise(0); 
END_IF 

IF Main.Errors.InMoldDryingErrors.TopMoldA.HeatingZone[6].PT100_WireBreak THEN 
Topmold_A_heating_zone_6_PT100_wirebreak.Raise(0); 
END_IF 

IF Main.Errors.InMoldDryingErrors.TopMoldA.HeatingZone[6].Thermal THEN 
Topmold_A_heating_zone_6_Thermal.Raise(0); 
END_IF 

IF Main.Errors.InMoldDryingErrors.TopMoldA.HeatingZone[6].PT100_TemperatureAboveMaximum THEN 
Topmold_A_heating_zone_6_temperature_above_250_degree_heating_element_switched_off.Raise(0); 
END_IF 

IF Main.Errors.InMoldDryingErrors.TopMoldA.HeatingZone[6].PT100_TemperatureTooHighWarn THEN 
Topmold_A_heating_zone_6_temperature_above_230_degree.Raise(0); 
END_IF 

IF Main.Errors.InMoldDryingErrors.BottomMoldA.HeatingZone[1].PT100_ConnectorNotConnected THEN 
Bottommold_A_heating_Zone_1_connector_not_connected.Raise(0); 
END_IF 

IF Main.Errors.InMoldDryingErrors.BottomMoldA.HeatingZone[1].PT100_HasWrongPosition THEN 
Bottommold_A_heating_Zone_1_PT100_wrong_position.Raise(0); 
END_IF 

IF Main.Errors.InMoldDryingErrors.BottomMoldA.HeatingZone[1].PT100_Loose THEN 
Bottommold_A_heating_Zone_1_PT100_loose.Raise(0); 
END_IF 

IF Main.Errors.InMoldDryingErrors.BottomMoldA.HeatingZone[1].PT100_NotInserted THEN 
Bottommold_A_heating_Zone_1_PT100_not_inserted.Raise(0); 
END_IF 

IF Main.Errors.InMoldDryingErrors.BottomMoldA.HeatingZone[1].PT100_TempAboveSetpoint THEN 
Bottommold_A_heating_Zone_1_Temperature_above_setpoint.Raise(0); 
END_IF 

IF Main.Errors.InMoldDryingErrors.BottomMoldA.HeatingZone[1].PT100_TempBelowSetpoint THEN 
Bottommold_A_heating_Zone_1_Temperature_below_setpoint.Raise(0); 
END_IF 

IF Main.Errors.InMoldDryingErrors.BottomMoldA.HeatingZone[1].PT100_WireBreak THEN 
Bottommold_A_heating_Zone_1_PT100_wirebreak.Raise(0); 
END_IF 

IF Main.Errors.InMoldDryingErrors.BottomMoldA.HeatingZone[1].Thermal THEN 
Bottommold_A_heating_Zone_1_Thermal.Raise(0); 
END_IF 

IF Main.Errors.InMoldDryingErrors.BottomMoldA.HeatingZone[1].PT100_TemperatureAboveMaximum THEN 
Bottommold_A_heating_zone_1_temperature_above_250_degree_heating_element_switched_off.Raise(0); 
END_IF 

IF Main.Errors.InMoldDryingErrors.BottomMoldA.HeatingZone[1].PT100_TemperatureTooHighWarn THEN 
Bottommold_A_heating_zone_1_temperature_above_230_degree.Raise(0); 
END_IF 

IF Main.Errors.InMoldDryingErrors.BottomMoldA.HeatingZone[2].PT100_ConnectorNotConnected THEN 
Bottommold_A_heating_Zone_2_connector_not_connected.Raise(0); 
END_IF 

IF Main.Errors.InMoldDryingErrors.BottomMoldA.HeatingZone[2].PT100_HasWrongPosition THEN 
Bottommold_A_heating_Zone_2_PT100_wrong_position.Raise(0); 
END_IF 

IF Main.Errors.InMoldDryingErrors.BottomMoldA.HeatingZone[2].PT100_Loose THEN 
Bottommold_A_heating_Zone_2_PT100_loose.Raise(0); 
END_IF 

IF Main.Errors.InMoldDryingErrors.BottomMoldA.HeatingZone[2].PT100_NotInserted THEN 
Bottommold_A_heating_Zone_2_PT100_not_inserted.Raise(0); 
END_IF 

IF Main.Errors.InMoldDryingErrors.BottomMoldA.HeatingZone[2].PT100_TempAboveSetpoint THEN 
Bottommold_A_heating_Zone_2_Temperature_above_setpoint.Raise(0); 
END_IF 

IF Main.Errors.InMoldDryingErrors.BottomMoldA.HeatingZone[2].PT100_TempBelowSetpoint THEN 
Bottommold_A_heating_Zone_2_Temperature_below_setpoint.Raise(0); 
END_IF 

IF Main.Errors.InMoldDryingErrors.BottomMoldA.HeatingZone[2].PT100_WireBreak THEN 
Bottommold_A_heating_Zone_2_PT100_wirebreak.Raise(0); 
END_IF 

IF Main.Errors.InMoldDryingErrors.BottomMoldA.HeatingZone[2].Thermal THEN 
Bottommold_A_heating_Zone_2_Thermal.Raise(0); 
END_IF 

IF Main.Errors.InMoldDryingErrors.BottomMoldA.HeatingZone[2].PT100_TemperatureAboveMaximum THEN 
Bottommold_A_heating_zone_2_temperature_above_250_degree_heating_element_switched_off.Raise(0); 
END_IF 

IF Main.Errors.InMoldDryingErrors.BottomMoldA.HeatingZone[2].PT100_TemperatureTooHighWarn THEN 
Bottommold_A_heating_zone_2_temperature_above_230_degree.Raise(0); 
END_IF 

IF Main.Errors.InMoldDryingErrors.BottomMoldA.HeatingZone[3].PT100_ConnectorNotConnected THEN 
Bottommold_A_heating_Zone_3_connector_not_connected.Raise(0); 
END_IF 

IF Main.Errors.InMoldDryingErrors.BottomMoldA.HeatingZone[3].PT100_HasWrongPosition THEN 
Bottommold_A_heating_Zone_3_PT100_wrong_position.Raise(0); 
END_IF 

IF Main.Errors.InMoldDryingErrors.BottomMoldA.HeatingZone[3].PT100_Loose  THEN 
Bottommold_A_heating_Zone_3_PT100_loose.Raise(0); 
END_IF 

IF Main.Errors.InMoldDryingErrors.BottomMoldA.HeatingZone[3].PT100_NotInserted THEN 
Bottommold_A_heating_Zone_3_PT100_not_inserted.Raise(0); 
END_IF 

IF Main.Errors.InMoldDryingErrors.BottomMoldA.HeatingZone[3].PT100_TempAboveSetpoint THEN 
Bottommold_A_heating_Zone_3_Temperature_above_setpoint.Raise(0); 
END_IF 

IF Main.Errors.InMoldDryingErrors.BottomMoldA.HeatingZone[3].PT100_TempBelowSetpoint THEN 
Bottommold_A_heating_Zone_3_Temperature_below_setpoint.Raise(0); 
END_IF 

IF Main.Errors.InMoldDryingErrors.BottomMoldA.HeatingZone[3].PT100_WireBreak THEN 
Bottommold_A_heating_Zone_3_PT100_wirebreak.Raise(0); 
END_IF 

IF Main.Errors.InMoldDryingErrors.BottomMoldA.HeatingZone[3].Thermal THEN 
Bottommold_A_heating_Zone_3_Thermal.Raise(0); 
END_IF 

IF Main.Errors.InMoldDryingErrors.BottomMoldA.HeatingZone[3].PT100_TemperatureAboveMaximum THEN 
Bottommold_A_heating_zone_3_temperature_above_250_degree_heating_element_switched_off.Raise(0); 
END_IF 

IF Main.Errors.InMoldDryingErrors.BottomMoldA.HeatingZone[3].PT100_TemperatureTooHighWarn THEN 
Bottommold_A_heating_zone_3_temperature_above_230_degree.Raise(0); 
END_IF 

IF Main.Errors.InMoldDryingErrors.BottomMoldA.HeatingZone[4].PT100_ConnectorNotConnected THEN 
Bottommold_A_heating_Zone_4_connector_not_connected.Raise(0); 
END_IF 

IF Main.Errors.InMoldDryingErrors.BottomMoldA.HeatingZone[4].PT100_HasWrongPosition THEN 
Bottommold_A_heating_Zone_4_PT100_wrong_position.Raise(0); 
END_IF 

IF Main.Errors.InMoldDryingErrors.BottomMoldA.HeatingZone[4].PT100_Loose THEN 
Bottommold_A_heating_Zone_4_PT100_loose.Raise(0); 
END_IF 

IF Main.Errors.InMoldDryingErrors.BottomMoldA.HeatingZone[4].PT100_NotInserted THEN 
Bottommold_A_heating_Zone_4_PT100_not_inserted.Raise(0); 
END_IF 

IF Main.Errors.InMoldDryingErrors.BottomMoldA.HeatingZone[4].PT100_TempAboveSetpoint THEN 
Bottommold_A_heating_Zone_4_Temperature_above_setpoint.Raise(0); 
END_IF 

IF Main.Errors.InMoldDryingErrors.BottomMoldA.HeatingZone[4].PT100_TempBelowSetpoint THEN 
Bottommold_A_heating_Zone_4_Temperature_below_setpoint.Raise(0); 
END_IF 

IF Main.Errors.InMoldDryingErrors.BottomMoldA.HeatingZone[4].PT100_WireBreak THEN 
Bottommold_A_heating_Zone_4_PT100_wirebreak.Raise(0); 
END_IF 

IF Main.Errors.InMoldDryingErrors.BottomMoldA.HeatingZone[4].Thermal THEN 
Bottommold_A_heating_Zone_4_Thermal.Raise(0); 
END_IF 

IF Main.Errors.InMoldDryingErrors.BottomMoldA.HeatingZone[4].PT100_TemperatureAboveMaximum THEN 
Bottommold_A_heating_zone_4_temperature_above_250_degree_heating_element_switched_off.Raise(0); 
END_IF 

IF Main.Errors.InMoldDryingErrors.BottomMoldA.HeatingZone[4].PT100_TemperatureTooHighWarn THEN 
Bottommold_A_heating_zone_4_temperature_above_230_degree.Raise(0); 
END_IF 

IF Main.Errors.InMoldDryingErrors.BottomMoldA.HeatingZone[5].PT100_ConnectorNotConnected THEN 
Bottommold_A_heating_Zone_5_connector_not_connected.Raise(0); 
END_IF 

IF Main.Errors.InMoldDryingErrors.BottomMoldA.HeatingZone[5].PT100_HasWrongPosition THEN 
Bottommold_A_heating_Zone_5_PT100_wrong_position.Raise(0); 
END_IF 

IF Main.Errors.InMoldDryingErrors.BottomMoldA.HeatingZone[5].PT100_Loose THEN 
Bottommold_A_heating_Zone_5_PT100_loose.Raise(0); 
END_IF 

IF Main.Errors.InMoldDryingErrors.BottomMoldA.HeatingZone[5].PT100_NotInserted THEN 
Bottommold_A_heating_Zone_5_PT100_not_inserted.Raise(0); 
END_IF 

IF Main.Errors.InMoldDryingErrors.BottomMoldA.HeatingZone[5].PT100_TempAboveSetpoint THEN 
Bottommold_A_heating_Zone_5_Temperature_above_setpoint.Raise(0); 
END_IF 

IF Main.Errors.InMoldDryingErrors.BottomMoldA.HeatingZone[5].PT100_TempBelowSetpoint THEN 
Bottommold_A_heating_Zone_5_Temperature_below_setpoint.Raise(0); 
END_IF 

IF Main.Errors.InMoldDryingErrors.BottomMoldA.HeatingZone[5].PT100_WireBreak THEN 
Bottommold_A_heating_Zone_5_PT100_wirebreak.Raise(0); 
END_IF 

IF Main.Errors.InMoldDryingErrors.BottomMoldA.HeatingZone[5].Thermal THEN 
Bottommold_A_heating_Zone_5_Thermal.Raise(0); 
END_IF 

IF Main.Errors.InMoldDryingErrors.BottomMoldA.HeatingZone[5].PT100_TemperatureAboveMaximum THEN 
Bottommold_A_heating_zone_5_temperature_above_250_degree_heating_element_switched_off.Raise(0); 
END_IF 

IF Main.Errors.InMoldDryingErrors.BottomMoldA.HeatingZone[5].PT100_TemperatureTooHighWarn THEN 
Bottommold_A_heating_zone_5_temperature_above_230_degree.Raise(0); 
END_IF 

IF Main.Errors.InMoldDryingErrors.BottomMoldA.HeatingZone[6].PT100_ConnectorNotConnected THEN 
Bottommold_A_heating_Zone_6_connector_not_connected.Raise(0); 
END_IF 

IF Main.Errors.InMoldDryingErrors.BottomMoldA.HeatingZone[6].PT100_HasWrongPosition THEN 
Bottommold_A_heating_Zone_6_PT100_wrong_position.Raise(0); 
END_IF 

IF Main.Errors.InMoldDryingErrors.BottomMoldA.HeatingZone[6].PT100_Loose THEN 
Bottommold_A_heating_Zone_6_PT100_loose.Raise(0); 
END_IF 

IF Main.Errors.InMoldDryingErrors.BottomMoldA.HeatingZone[6].PT100_NotInserted THEN 
Bottommold_A_heating_Zone_6_PT100_not_inserted.Raise(0); 
END_IF 

IF Main.Errors.InMoldDryingErrors.BottomMoldA.HeatingZone[6].PT100_TempAboveSetpoint THEN 
Bottommold_A_heating_Zone_6_Temperature_above_setpoint.Raise(0); 
END_IF 

IF Main.Errors.InMoldDryingErrors.BottomMoldA.HeatingZone[6].PT100_TempBelowSetpoint THEN 
Bottommold_A_heating_Zone_6_Temperature_below_setpoint.Raise(0); 
END_IF 

IF Main.Errors.InMoldDryingErrors.BottomMoldA.HeatingZone[6].PT100_WireBreak THEN 
Bottommold_A_heating_Zone_6_PT100_wirebreak.Raise(0); 
END_IF 

IF Main.Errors.InMoldDryingErrors.BottomMoldA.HeatingZone[6].Thermal THEN 
Bottommold_A_heating_Zone_6_Thermal.Raise(0); 
END_IF 

IF Main.Errors.InMoldDryingErrors.BottomMoldA.HeatingZone[6].PT100_TemperatureAboveMaximum THEN 
Bottommold_A_heating_zone_6_temperature_above_250_degree_heating_element_switched_off.Raise(0); 
END_IF 

IF Main.Errors.InMoldDryingErrors.TopMoldB.TmDidNotReachBmPosTimeOut THEN 
Top_mold_B_timed_out_Did_not_reach_bottommold_position_in_time.Raise(0); 
END_IF 

IF Main.Errors.InMoldDryingErrors.TopMoldB.Hydraulic.BallufError THEN 
Top_mold_B_error_on_balluf.Raise(0); 
END_IF 

IF Main.Errors.InMoldDryingErrors.TopMoldB.Hydraulic.IsMovingWithoutActivation THEN 
Top_mold_B_is_moving_without_activation.Raise(0); 
END_IF 

IF Main.Errors.InMoldDryingErrors.BottomMoldA.HeatingZone[6].PT100_TemperatureTooHighWarn THEN 
Bottommold_A_heating_zone_6_temperature_above_230_degree.Raise(0); 
END_IF 

IF Main.Errors.InMoldDryingErrors.TopMoldB.HeatingZone[1].PT100_ConnectorNotConnected THEN 
Topmold_B_heating_Zone_1_connector_not_connected.Raise(0); 
END_IF 

IF Main.Errors.InMoldDryingErrors.TopMoldB.HeatingZone[1].PT100_HasWrongPosition THEN 
Topmold_B_heating_Zone_1_PT100_wrong_position.Raise(0); 
END_IF 

IF Main.Errors.InMoldDryingErrors.TopMoldB.HeatingZone[1].PT100_Loose THEN 
Topmold_B_heating_Zone_1_PT100_loose.Raise(0); 
END_IF 

IF Main.Errors.InMoldDryingErrors.TopMoldB.HeatingZone[1].PT100_NotInserted THEN 
Topmold_B_heating_Zone_1_PT100_not_inserted.Raise(0); 
END_IF 

IF Main.Errors.InMoldDryingErrors.TopMoldB.HeatingZone[1].PT100_TempAboveSetpoint THEN 
Topmold_B_heating_Zone_1_Temperature_above_setpoint.Raise(0); 
END_IF 

IF Main.Errors.InMoldDryingErrors.TopMoldB.HeatingZone[1].PT100_TempBelowSetpoint THEN 
Topmold_B_heating_Zone_1_Temperature_below_setpoint.Raise(0); 
END_IF 

IF Main.Errors.InMoldDryingErrors.TopMoldB.HeatingZone[1].PT100_WireBreak THEN 
Topmold_B_heating_Zone_1_PT100_wirebreak.Raise(0); 
END_IF 

IF Main.Errors.InMoldDryingErrors.TopMoldB.HeatingZone[1].Thermal THEN 
Topmold_B_heating_Zone_1_Thermal.Raise(0); 
END_IF 

IF Main.Errors.InMoldDryingErrors.TopMoldB.HeatingZone[1].PT100_TemperatureAboveMaximum THEN 
Topmold_B_heating_zone_1_temperature_above_250_degree_heating_element_switched_off.Raise(0); 
END_IF 

IF Main.Errors.InMoldDryingErrors.TopMoldB.HeatingZone[1].PT100_TemperatureTooHighWarn THEN 
Topmold_B_heating_zone_1_temperature_above_230_degree.Raise(0); 
END_IF 

IF Main.Errors.InMoldDryingErrors.TopMoldB.HeatingZone[2].PT100_ConnectorNotConnected THEN 
Topmold_B_heating_Zone_2_connector_not_connected.Raise(0); 
END_IF 

IF Main.Errors.InMoldDryingErrors.TopMoldB.HeatingZone[2].PT100_HasWrongPosition THEN 
Topmold_B_heating_Zone_2_PT100_wrong_position.Raise(0); 
END_IF 

IF Main.Errors.InMoldDryingErrors.TopMoldB.HeatingZone[2].PT100_Loose THEN 
Topmold_B_heating_Zone_2_PT100_loose.Raise(0); 
END_IF 

IF Main.Errors.InMoldDryingErrors.TopMoldB.HeatingZone[2].PT100_NotInserted THEN 
Topmold_B_heating_Zone_2_PT100_not_inserted.Raise(0); 
END_IF 

IF Main.Errors.InMoldDryingErrors.TopMoldB.HeatingZone[2].PT100_TempAboveSetpoint THEN 
Topmold_B_heating_Zone_2_Temperature_above_setpoint.Raise(0); 
END_IF 

IF Main.Errors.InMoldDryingErrors.TopMoldB.HeatingZone[2].PT100_TempBelowSetpoint THEN 
Topmold_B_heating_Zone_2_Temperature_below_setpoint.Raise(0); 
END_IF 

IF Main.Errors.InMoldDryingErrors.TopMoldB.HeatingZone[2].PT100_WireBreak THEN 
Topmold_B_heating_Zone_2_PT100_wirebreak.Raise(0); 
END_IF 

IF Main.Errors.InMoldDryingErrors.TopMoldB.HeatingZone[2].Thermal THEN 
Topmold_B_heating_Zone_2_Thermal.Raise(0); 
END_IF 

IF Main.Errors.InMoldDryingErrors.TopMoldB.HeatingZone[2].PT100_TemperatureAboveMaximum THEN 
Topmold_B_heating_zone_2_temperature_above_250_degree_heating_element_switched_off.Raise(0); 
END_IF 

IF Main.Errors.InMoldDryingErrors.TopMoldB.HeatingZone[2].PT100_TemperatureTooHighWarn THEN 
Topmold_B_heating_zone_2_temperature_above_230_degree.Raise(0); 
END_IF 

IF Main.Errors.InMoldDryingErrors.TopMoldB.HeatingZone[3].PT100_ConnectorNotConnected THEN 
Topmold_B_heating_Zone_3_connector_not_connected.Raise(0); 
END_IF 

IF Main.Errors.InMoldDryingErrors.TopMoldB.HeatingZone[3].PT100_HasWrongPosition THEN 
Topmold_B_heating_Zone_3_PT100_wrong_position.Raise(0); 
END_IF 

IF Main.Errors.InMoldDryingErrors.TopMoldB.HeatingZone[3].PT100_Loose THEN 
Topmold_B_heating_Zone_3_PT100_loose.Raise(0); 
END_IF 

IF Main.Errors.InMoldDryingErrors.TopMoldB.HeatingZone[3].PT100_NotInserted THEN 
Topmold_B_heating_Zone_3_PT100_not_inserted.Raise(0); 
END_IF 

IF Main.Errors.InMoldDryingErrors.TopMoldB.HeatingZone[3].PT100_TempAboveSetpoint THEN 
Topmold_B_heating_Zone_3_Temperature_above_setpoint.Raise(0); 
END_IF 

IF Main.Errors.InMoldDryingErrors.TopMoldB.HeatingZone[3].PT100_TempBelowSetpoint THEN 
Topmold_B_heating_Zone_3_Temperature_below_setpoint.Raise(0); 
END_IF 

IF Main.Errors.InMoldDryingErrors.TopMoldB.HeatingZone[3].PT100_WireBreak THEN 
Topmold_B_heating_Zone_3_PT100_wirebreak.Raise(0); 
END_IF 

IF Main.Errors.InMoldDryingErrors.TopMoldB.HeatingZone[3].Thermal THEN 
Topmold_B_heating_Zone_3_Thermal.Raise(0); 
END_IF 

IF Main.Errors.InMoldDryingErrors.TopMoldB.HeatingZone[3].PT100_TemperatureAboveMaximum THEN 
Topmold_B_heating_zone_3_temperature_above_250_degree_heating_element_switched_off.Raise(0); 
END_IF 

IF Main.Errors.InMoldDryingErrors.TopMoldB.HeatingZone[3].PT100_TemperatureTooHighWarn THEN 
Topmold_B_heating_zone_3_temperature_above_230_degree.Raise(0); 
END_IF 

IF Main.Errors.InMoldDryingErrors.TopMoldB.HeatingZone[4].PT100_ConnectorNotConnected THEN 
Topmold_B_heating_Zone_4_connector_not_connected.Raise(0); 
END_IF 

IF Main.Errors.InMoldDryingErrors.TopMoldB.HeatingZone[4].PT100_HasWrongPosition THEN 
Topmold_B_heating_Zone_4_PT100_wrong_position.Raise(0); 
END_IF 

IF Main.Errors.InMoldDryingErrors.TopMoldB.HeatingZone[4].PT100_Loose THEN 
Topmold_B_heating_Zone_4_PT100_loose.Raise(0); 
END_IF 

IF Main.Errors.InMoldDryingErrors.TopMoldB.HeatingZone[4].PT100_NotInserted THEN 
Topmold_B_heating_Zone_4_PT100_not_inserted.Raise(0); 
END_IF 

IF Main.Errors.InMoldDryingErrors.TopMoldB.HeatingZone[4].PT100_TempAboveSetpoint THEN 
Topmold_B_heating_Zone_4_Temperature_above_setpoint.Raise(0); 
END_IF 

IF Main.Errors.InMoldDryingErrors.TopMoldB.HeatingZone[4].PT100_TempBelowSetpoint THEN 
Topmold_B_heating_Zone_4_Temperature_below_setpoint.Raise(0); 
END_IF 

IF Main.Errors.InMoldDryingErrors.TopMoldB.HeatingZone[4].PT100_WireBreak THEN 
Topmold_B_heating_Zone_4_PT100_wirebreak.Raise(0); 
END_IF 

IF Main.Errors.InMoldDryingErrors.TopMoldB.HeatingZone[4].Thermal THEN 
Topmold_B_heating_Zone_4_Thermal.Raise(0); 
END_IF 

IF Main.Errors.InMoldDryingErrors.TopMoldB.HeatingZone[4].PT100_TemperatureAboveMaximum THEN 
Topmold_B_heating_zone_4_temperature_above_250_degree_heating_element_switched_off.Raise(0); 
END_IF 

IF Main.Errors.InMoldDryingErrors.TopMoldB.HeatingZone[4].PT100_TemperatureTooHighWarn THEN 
Topmold_B_heating_zone_4_temperature_above_230_degree.Raise(0); 
END_IF 

IF Main.Errors.InMoldDryingErrors.TopMoldB.HeatingZone[5].PT100_ConnectorNotConnected THEN 
Topmold_B_heating_Zone_5_connector_not_connected.Raise(0); 
END_IF 

IF Main.Errors.InMoldDryingErrors.TopMoldB.HeatingZone[5].PT100_HasWrongPosition THEN 
Topmold_B_heating_Zone_5_PT100_wrong_position.Raise(0); 
END_IF 

IF Main.Errors.InMoldDryingErrors.TopMoldB.HeatingZone[5].PT100_Loose THEN 
Topmold_B_heating_Zone_5_PT100_loose.Raise(0); 
END_IF 

IF Main.Errors.InMoldDryingErrors.TopMoldB.HeatingZone[5].PT100_NotInserted THEN 
Topmold_B_heating_Zone_5_PT100_not_inserted.Raise(0); 
END_IF 

IF Main.Errors.InMoldDryingErrors.TopMoldB.HeatingZone[5].PT100_TempAboveSetpoint THEN 
Topmold_B_heating_Zone_5_Temperature_above_setpoint.Raise(0); 
END_IF 

IF Main.Errors.InMoldDryingErrors.TopMoldB.HeatingZone[5].PT100_TempBelowSetpoint THEN 
Topmold_B_heating_Zone_5_Temperature_below_setpoint.Raise(0); 
END_IF 

IF Main.Errors.InMoldDryingErrors.TopMoldB.HeatingZone[5].PT100_WireBreak THEN 
Topmold_B_heating_Zone_5_PT100_wirebreak.Raise(0); 
END_IF 

IF Main.Errors.InMoldDryingErrors.TopMoldB.HeatingZone[5].Thermal THEN 
Topmold_B_heating_Zone_5_Thermal.Raise(0); 
END_IF 

IF Main.Errors.InMoldDryingErrors.TopMoldB.HeatingZone[5].PT100_TemperatureAboveMaximum THEN 
Topmold_B_heating_zone_5_temperature_above_250_degree_heating_element_switched_off.Raise(0); 
END_IF 

IF Main.Errors.InMoldDryingErrors.TopMoldB.HeatingZone[5].PT100_TemperatureTooHighWarn THEN 
Topmold_B_heating_zone_5_temperature_above_230_degree.Raise(0); 
END_IF 

IF Main.Errors.InMoldDryingErrors.TopMoldB.HeatingZone[6].PT100_ConnectorNotConnected THEN 
Topmold_B_heating_Zone_6_connector_not_connected.Raise(0); 
END_IF 

